FUNCTION_BLOCK "Graph_Sequence"   // FB265, GRAPH
VERSION : 0.1
// stored: AcknowledgeErrorsRequired true, AutoNumber true, GraphVersion 6.0, InitialValuesAcquisition false, IsIECCheckEnabled false, LanguageInNetworks LAD, LockOperatingMode false, PermanentILProcessingInMANMode false, SetENOAutomatically false, SkipSteps true, UDAEnableTagReadback false, WithAlarmHandling true
   // inherited from GRAPH_BASE
   VAR
      OFF_SQ_BASE : Bool;
   END_VAR
   VAR_INPUT
      ACK_EF { ExternalAccessible := 'False'; ExternalVisible := 'False'; ExternalWritable := 'False'} : Bool := false;   // Acknowledge all errors and faults
      INIT_SQ { ExternalAccessible := 'False'; ExternalVisible := 'False'; ExternalWritable := 'False'} : Bool := false;   // Set sequence to initial state
      stepTimeOutTime : Time;
      iInstance_Index : DInt;
   END_VAR
   VAR_IN_OUT
      funcGrp : "typeCaCgFg";   // Funktionsgruppe / Function Group
      fgControlGeneral_1 : "typeFgControlGeneral";   // Funktionsgruppe Steuerung / Function group control system
      ioJobSelect : Int;
   END_VAR
   VAR
      instGraphEval { ExternalAccessible := 'False'; ExternalVisible := 'False'; ExternalWritable := 'False'} : "GraphEvaluation";   // FG Laser 1: S7-Graph Auswertung / FG laser 1: S7-Graph evaluation
      fgControlGeneral { ExternalAccessible := 'False'; ExternalVisible := 'False'; ExternalWritable := 'False'} : "typeFgControlGeneral";   // Funktionsgruppe Steuerung / Function group control system
      stepTimeOut : Bool;
   END_VAR
BEGIN
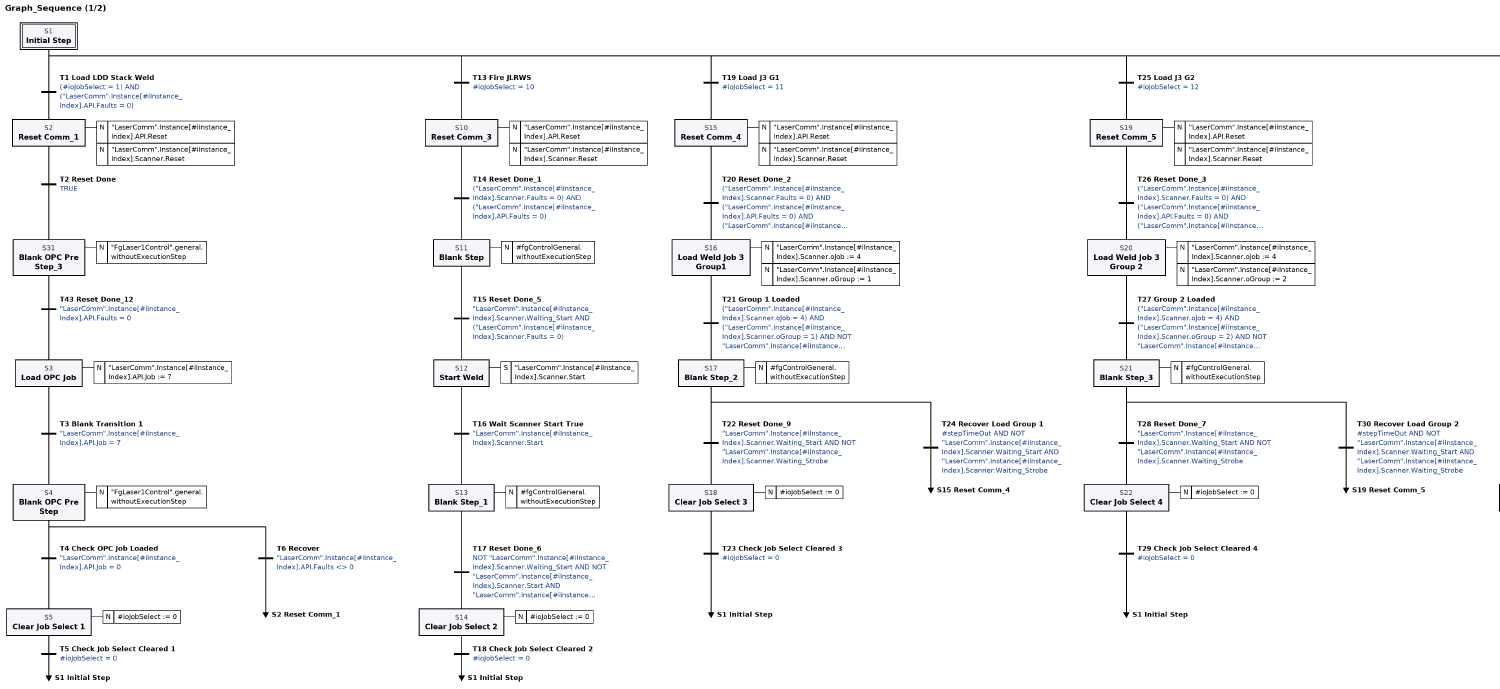
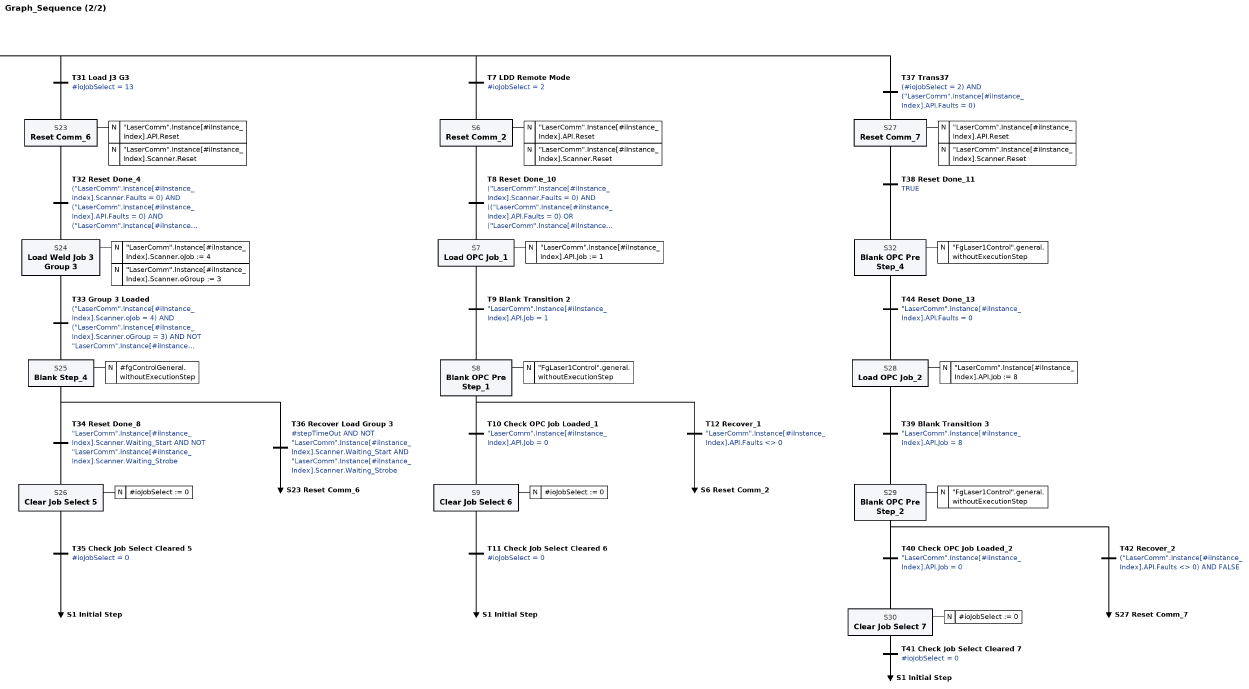
   // sequencer 1: Weld Graph Sequences
   INITIAL_STEP "Initial Step":   // S1, max time T#10S, warning time T#7S
   END_STEP
   TRANSITION "Load LDD Stack Weld" FROM "Initial Step" TO "Reset Comm_1"   // T1
      := (#ioJobSelect = 1) AND ("LaserComm".Instance[#iInstance_Index].API.Faults = 0);
   END_TRANSITION
   TRANSITION "Fire JLRWS" FROM "Initial Step" TO "Reset Comm_3"   // T13
      := #ioJobSelect = 10;
   END_TRANSITION
   TRANSITION "Load J3 G1" FROM "Initial Step" TO "Reset Comm_4"   // T19
      := #ioJobSelect = 11;
   END_TRANSITION
   TRANSITION "Load J3 G2" FROM "Initial Step" TO "Reset Comm_5"   // T25
      := #ioJobSelect = 12;
   END_TRANSITION
   TRANSITION "Load J3 G3" FROM "Initial Step" TO "Reset Comm_6"   // T31
      := #ioJobSelect = 13;
   END_TRANSITION
   TRANSITION "LDD Remote Mode" FROM "Initial Step" TO "Reset Comm_2"   // T7
      := #ioJobSelect = 2;
   END_TRANSITION
   TRANSITION Trans37 FROM "Initial Step" TO "Reset Comm_7"   // T37
      := (#ioJobSelect = 2) AND ("LaserComm".Instance[#iInstance_Index].API.Faults = 0);
   END_TRANSITION
   STEP "Reset Comm_1":   // S2, max time T#10S, warning time T#7S
      supervision V := #stepTimeOut;
              N    "LaserComm".Instance[#iInstance_Index].API.Reset
              N    "LaserComm".Instance[#iInstance_Index].Scanner.Reset
   END_STEP
   TRANSITION "Reset Done" FROM "Reset Comm_1" TO "Blank OPC Pre Step_3"   // T2
      := TRUE;
   END_TRANSITION
   STEP "Blank Step":   // S11, max time T#10S, warning time T#7S
      supervision V := #stepTimeOut;
              N    #fgControlGeneral.withoutExecutionStep
   END_STEP
   TRANSITION "Reset Done_5" FROM "Blank Step" TO "Start Weld"   // T15
      := "LaserComm".Instance[#iInstance_Index].Scanner.Waiting_Start AND ("LaserComm".Instance[#iInstance_Index].Scanner.Faults = 0);
   END_TRANSITION
   STEP "Clear Job Select 4":   // S22, max time T#10S, warning time T#7S
      supervision V := #stepTimeOut;
      // Clear Job Select
              N    #ioJobSelect := 0
   END_STEP
   TRANSITION "Check Job Select Cleared 4" FROM "Clear Job Select 4" TO "Initial Step"   // T29, jump: Check Jo Select Cleared
      := #ioJobSelect = 0;
   END_TRANSITION
   STEP "Clear Job Select 5":   // S26, max time T#10S, warning time T#7S
      supervision V := #stepTimeOut;
      // Clear Job Select
              N    #ioJobSelect := 0
   END_STEP
   TRANSITION "Check Job Select Cleared 5" FROM "Clear Job Select 5" TO "Initial Step"   // T35, jump: Check Jo Select Cleared
      := #ioJobSelect = 0;
   END_TRANSITION
   STEP "Load Weld Job 3 Group 3":   // S24, max time T#10S, warning time T#7S
      supervision V := #stepTimeOut;
              N    "LaserComm".Instance[#iInstance_Index].Scanner.oJob := 4
              N    "LaserComm".Instance[#iInstance_Index].Scanner.oGroup := 3
   END_STEP
   TRANSITION "Group 3 Loaded" FROM "Load Weld Job 3 Group 3" TO "Blank Step_4"   // T33
      := ("LaserComm".Instance[#iInstance_Index].Scanner.oJob = 4) AND ("LaserComm".Instance[#iInstance_Index].Scanner.oGroup = 3) AND NOT "LaserComm".Instance[#iInstance_Index].Scanner.Waiting_Strobe;
   END_TRANSITION
   STEP "Load OPC Job":   // S3, max time T#10S, warning time T#7S
      supervision V := #stepTimeOut;
              N    "LaserComm".Instance[#iInstance_Index].API.Job := 7
   END_STEP
   TRANSITION "Blank Transition 1" FROM "Load OPC Job" TO "Blank OPC Pre Step"   // T3
      := "LaserComm".Instance[#iInstance_Index].API.Job = 7;
   END_TRANSITION
   STEP "Blank OPC Pre Step":   // S4, max time T#10S, warning time T#7S
      supervision V := #stepTimeOut;
              N    "FgLaser1Control".general.withoutExecutionStep
   END_STEP
   TRANSITION "Check OPC Job Loaded" FROM "Blank OPC Pre Step" TO "Clear Job Select 1"   // T4
      := "LaserComm".Instance[#iInstance_Index].API.Job = 0;
   END_TRANSITION
   TRANSITION Recover FROM "Blank OPC Pre Step" TO "Reset Comm_1"   // T6, jump
      := "LaserComm".Instance[#iInstance_Index].API.Faults <> 0;
   END_TRANSITION
   STEP "Clear Job Select 1":   // S5, max time T#10S, warning time T#7S
      supervision V := #stepTimeOut;
      // Clear Job Select
              N    #ioJobSelect := 0
   END_STEP
   TRANSITION "Check Job Select Cleared 1" FROM "Clear Job Select 1" TO "Initial Step"   // T5, jump: Check Jo Select Cleared
      := #ioJobSelect = 0;
   END_TRANSITION
   STEP "Blank Step_1":   // S13, max time T#10S, warning time T#7S
      supervision V := #stepTimeOut;
              N    #fgControlGeneral.withoutExecutionStep
   END_STEP
   TRANSITION "Reset Done_6" FROM "Blank Step_1" TO "Clear Job Select 2"   // T17
      := NOT "LaserComm".Instance[#iInstance_Index].Scanner.Waiting_Start AND NOT "LaserComm".Instance[#iInstance_Index].Scanner.Start AND "LaserComm".Instance[#iInstance_Index].Scanner.Waiting_Strobe AND ("LaserComm".Instance[#iInstance_Index].Scanner.Faults = 0);
   END_TRANSITION
   STEP "Reset Comm_3":   // S10, max time T#10S, warning time T#7S
      supervision V := #stepTimeOut;
              N    "LaserComm".Instance[#iInstance_Index].API.Reset
              N    "LaserComm".Instance[#iInstance_Index].Scanner.Reset
   END_STEP
   TRANSITION "Reset Done_1" FROM "Reset Comm_3" TO "Blank Step"   // T14
      := ("LaserComm".Instance[#iInstance_Index].Scanner.Faults = 0) AND ("LaserComm".Instance[#iInstance_Index].API.Faults = 0);
   END_TRANSITION
   STEP "Load Weld Job 3 Group1":   // S16, max time T#10S, warning time T#7S
      supervision V := #stepTimeOut;
              N    "LaserComm".Instance[#iInstance_Index].Scanner.oJob := 4
              N    "LaserComm".Instance[#iInstance_Index].Scanner.oGroup := 1
   END_STEP
   TRANSITION "Group 1 Loaded" FROM "Load Weld Job 3 Group1" TO "Blank Step_2"   // T21
      := ("LaserComm".Instance[#iInstance_Index].Scanner.oJob = 4) AND ("LaserComm".Instance[#iInstance_Index].Scanner.oGroup = 1) AND NOT "LaserComm".Instance[#iInstance_Index].Scanner.Waiting_Strobe;
   END_TRANSITION
   STEP "Load Weld Job 3 Group 2":   // S20, max time T#10S, warning time T#7S
      supervision V := #stepTimeOut;
              N    "LaserComm".Instance[#iInstance_Index].Scanner.oJob := 4
              N    "LaserComm".Instance[#iInstance_Index].Scanner.oGroup := 2
   END_STEP
   TRANSITION "Group 2 Loaded" FROM "Load Weld Job 3 Group 2" TO "Blank Step_3"   // T27
      := ("LaserComm".Instance[#iInstance_Index].Scanner.oJob = 4) AND ("LaserComm".Instance[#iInstance_Index].Scanner.oGroup = 2) AND NOT "LaserComm".Instance[#iInstance_Index].Scanner.Waiting_Strobe;
   END_TRANSITION
   STEP "Reset Comm_4":   // S15, max time T#10S, warning time T#7S
      supervision V := #stepTimeOut;
              N    "LaserComm".Instance[#iInstance_Index].API.Reset
              N    "LaserComm".Instance[#iInstance_Index].Scanner.Reset
   END_STEP
   TRANSITION "Reset Done_2" FROM "Reset Comm_4" TO "Load Weld Job 3 Group1"   // T20
      := ("LaserComm".Instance[#iInstance_Index].Scanner.Faults = 0) AND ("LaserComm".Instance[#iInstance_Index].API.Faults = 0) AND ("LaserComm".Instance[#iInstance_Index].Scanner.oJob = 0) AND ("LaserComm".Instance[#iInstance_Index].Scanner.oGroup = 0) AND "LaserComm".Instance[#iInstance_Index].Scanner.Waiting_Strobe;
   END_TRANSITION
   STEP "Reset Comm_5":   // S19, max time T#10S, warning time T#7S
      supervision V := #stepTimeOut;
              N    "LaserComm".Instance[#iInstance_Index].API.Reset
              N    "LaserComm".Instance[#iInstance_Index].Scanner.Reset
   END_STEP
   TRANSITION "Reset Done_3" FROM "Reset Comm_5" TO "Load Weld Job 3 Group 2"   // T26
      := ("LaserComm".Instance[#iInstance_Index].Scanner.Faults = 0) AND ("LaserComm".Instance[#iInstance_Index].API.Faults = 0) AND ("LaserComm".Instance[#iInstance_Index].Scanner.oJob = 0) AND ("LaserComm".Instance[#iInstance_Index].Scanner.oGroup = 0);
   END_TRANSITION
   STEP "Reset Comm_6":   // S23, max time T#10S, warning time T#7S
      supervision V := #stepTimeOut;
              N    "LaserComm".Instance[#iInstance_Index].API.Reset
              N    "LaserComm".Instance[#iInstance_Index].Scanner.Reset
   END_STEP
   TRANSITION "Reset Done_4" FROM "Reset Comm_6" TO "Load Weld Job 3 Group 3"   // T32
      := ("LaserComm".Instance[#iInstance_Index].Scanner.Faults = 0) AND ("LaserComm".Instance[#iInstance_Index].API.Faults = 0) AND ("LaserComm".Instance[#iInstance_Index].Scanner.oJob = 0) AND ("LaserComm".Instance[#iInstance_Index].Scanner.oGroup = 0);
   END_TRANSITION
   STEP "Clear Job Select 3":   // S18, max time T#10S, warning time T#7S
      supervision V := #stepTimeOut;
      // Clear Job Select
              N    #ioJobSelect := 0
   END_STEP
   TRANSITION "Check Job Select Cleared 3" FROM "Clear Job Select 3" TO "Initial Step"   // T23, jump: Check Jo Select Cleared
      := #ioJobSelect = 0;
   END_TRANSITION
   STEP "Clear Job Select 2":   // S14, max time T#10S, warning time T#7S
      supervision V := #stepTimeOut;
      // Clear Job Select
              N    #ioJobSelect := 0
   END_STEP
   TRANSITION "Check Job Select Cleared 2" FROM "Clear Job Select 2" TO "Initial Step"   // T18, jump: Check Jo Select Cleared
      := #ioJobSelect = 0;
   END_TRANSITION
   STEP "Start Weld":   // S12, max time T#10S, warning time T#7S
      supervision V := #stepTimeOut;
              S    "LaserComm".Instance[#iInstance_Index].Scanner.Start
   END_STEP
   TRANSITION "Wait Scanner Start True" FROM "Start Weld" TO "Blank Step_1"   // T16
      := "LaserComm".Instance[#iInstance_Index].Scanner.Start;
   END_TRANSITION
   STEP "Blank Step_3":   // S21, max time T#10S, warning time T#7S
      supervision V := #stepTimeOut;
              N    #fgControlGeneral.withoutExecutionStep
   END_STEP
   TRANSITION "Reset Done_7" FROM "Blank Step_3" TO "Clear Job Select 4"   // T28
      := "LaserComm".Instance[#iInstance_Index].Scanner.Waiting_Start AND NOT "LaserComm".Instance[#iInstance_Index].Scanner.Waiting_Strobe;
   END_TRANSITION
   TRANSITION "Recover Load Group 2" FROM "Blank Step_3" TO "Reset Comm_5"   // T30, jump
      := #stepTimeOut AND NOT "LaserComm".Instance[#iInstance_Index].Scanner.Waiting_Start AND "LaserComm".Instance[#iInstance_Index].Scanner.Waiting_Strobe;
   END_TRANSITION
   STEP "Blank Step_4":   // S25, max time T#10S, warning time T#7S
      supervision V := #stepTimeOut;
              N    #fgControlGeneral.withoutExecutionStep
   END_STEP
   TRANSITION "Reset Done_8" FROM "Blank Step_4" TO "Clear Job Select 5"   // T34
      := "LaserComm".Instance[#iInstance_Index].Scanner.Waiting_Start AND NOT "LaserComm".Instance[#iInstance_Index].Scanner.Waiting_Strobe;
   END_TRANSITION
   TRANSITION "Recover Load Group 3" FROM "Blank Step_4" TO "Reset Comm_6"   // T36, jump
      := #stepTimeOut AND NOT "LaserComm".Instance[#iInstance_Index].Scanner.Waiting_Start AND "LaserComm".Instance[#iInstance_Index].Scanner.Waiting_Strobe;
   END_TRANSITION
   STEP "Blank Step_2":   // S17, max time T#10S, warning time T#7S
      supervision V := #stepTimeOut;
              N    #fgControlGeneral.withoutExecutionStep
   END_STEP
   TRANSITION "Reset Done_9" FROM "Blank Step_2" TO "Clear Job Select 3"   // T22
      := "LaserComm".Instance[#iInstance_Index].Scanner.Waiting_Start AND NOT "LaserComm".Instance[#iInstance_Index].Scanner.Waiting_Strobe;
   END_TRANSITION
   TRANSITION "Recover Load Group 1" FROM "Blank Step_2" TO "Reset Comm_4"   // T24, jump
      := #stepTimeOut AND NOT "LaserComm".Instance[#iInstance_Index].Scanner.Waiting_Start AND "LaserComm".Instance[#iInstance_Index].Scanner.Waiting_Strobe;
   END_TRANSITION
   STEP "Reset Comm_2":   // S6, max time T#10S, warning time T#7S
      supervision V := #stepTimeOut;
              N    "LaserComm".Instance[#iInstance_Index].API.Reset
              N    "LaserComm".Instance[#iInstance_Index].Scanner.Reset
   END_STEP
   TRANSITION "Reset Done_10" FROM "Reset Comm_2" TO "Load OPC Job_1"   // T8
      := ("LaserComm".Instance[#iInstance_Index].Scanner.Faults = 0) AND (("LaserComm".Instance[#iInstance_Index].API.Faults = 0) OR ("LaserComm".Instance[#iInstance_Index].API.Faults = 64));
   END_TRANSITION
   STEP "Load OPC Job_1":   // S7, max time T#10S, warning time T#7S
      supervision V := #stepTimeOut;
              N    "LaserComm".Instance[#iInstance_Index].API.Job := 1
   END_STEP
   TRANSITION "Blank Transition 2" FROM "Load OPC Job_1" TO "Blank OPC Pre Step_1"   // T9
      := "LaserComm".Instance[#iInstance_Index].API.Job = 1;
   END_TRANSITION
   STEP "Blank OPC Pre Step_1":   // S8, max time T#10S, warning time T#7S
      supervision V := #stepTimeOut;
              N    "FgLaser1Control".general.withoutExecutionStep
   END_STEP
   TRANSITION "Check OPC Job Loaded_1" FROM "Blank OPC Pre Step_1" TO "Clear Job Select 6"   // T10
      := "LaserComm".Instance[#iInstance_Index].API.Job = 0;
   END_TRANSITION
   TRANSITION Recover_1 FROM "Blank OPC Pre Step_1" TO "Reset Comm_2"   // T12, jump
      := "LaserComm".Instance[#iInstance_Index].API.Faults <> 0;
   END_TRANSITION
   STEP "Clear Job Select 6":   // S9, max time T#10S, warning time T#7S
      supervision V := #stepTimeOut;
      // Clear Job Select
              N    #ioJobSelect := 0
   END_STEP
   TRANSITION "Check Job Select Cleared 6" FROM "Clear Job Select 6" TO "Initial Step"   // T11, jump: Check Jo Select Cleared
      := #ioJobSelect = 0;
   END_TRANSITION
   STEP "Reset Comm_7":   // S27, max time T#10S, warning time T#7S
      supervision V := #stepTimeOut;
              N    "LaserComm".Instance[#iInstance_Index].API.Reset
              N    "LaserComm".Instance[#iInstance_Index].Scanner.Reset
   END_STEP
   TRANSITION "Reset Done_11" FROM "Reset Comm_7" TO "Blank OPC Pre Step_4"   // T38
      := TRUE;
   END_TRANSITION
   STEP "Load OPC Job_2":   // S28, max time T#10S, warning time T#7S
      supervision V := #stepTimeOut;
              N    "LaserComm".Instance[#iInstance_Index].API.Job := 8
   END_STEP
   TRANSITION "Blank Transition 3" FROM "Load OPC Job_2" TO "Blank OPC Pre Step_2"   // T39
      := "LaserComm".Instance[#iInstance_Index].API.Job = 8;
   END_TRANSITION
   STEP "Blank OPC Pre Step_2":   // S29, max time T#10S, warning time T#7S
      supervision V := #stepTimeOut;
              N    "FgLaser1Control".general.withoutExecutionStep
   END_STEP
   TRANSITION "Check OPC Job Loaded_2" FROM "Blank OPC Pre Step_2" TO "Clear Job Select 7"   // T40
      := "LaserComm".Instance[#iInstance_Index].API.Job = 0;
   END_TRANSITION
   TRANSITION Recover_2 FROM "Blank OPC Pre Step_2" TO "Reset Comm_7"   // T42, jump
      := ("LaserComm".Instance[#iInstance_Index].API.Faults <> 0) AND FALSE;
   END_TRANSITION
   STEP "Clear Job Select 7":   // S30, max time T#10S, warning time T#7S
      supervision V := #stepTimeOut;
      // Clear Job Select
              N    #ioJobSelect := 0
   END_STEP
   TRANSITION "Check Job Select Cleared 7" FROM "Clear Job Select 7" TO "Initial Step"   // T41, jump: Check Jo Select Cleared
      := #ioJobSelect = 0;
   END_TRANSITION
   STEP "Blank OPC Pre Step_3":   // S31, max time T#10S, warning time T#7S
      supervision V := #stepTimeOut;
              N    "FgLaser1Control".general.withoutExecutionStep
   END_STEP
   TRANSITION "Reset Done_12" FROM "Blank OPC Pre Step_3" TO "Load OPC Job"   // T43
      := "LaserComm".Instance[#iInstance_Index].API.Faults = 0;
   END_TRANSITION
   STEP "Blank OPC Pre Step_4":   // S32, max time T#10S, warning time T#7S
      supervision V := #stepTimeOut;
              N    "FgLaser1Control".general.withoutExecutionStep
   END_STEP
   TRANSITION "Reset Done_13" FROM "Blank OPC Pre Step_4" TO "Load OPC Job_2"   // T44
      := "LaserComm".Instance[#iInstance_Index].API.Faults = 0;
   END_TRANSITION

   // permanent post-instructions
   NETWORK 1
      #instGraphEval(rtData := #RT_DATA,   // "GraphEvaluation"
                     timeOutTime := #stepTimeOutTime,
                     funcGrp := #funcGrp,
                     fgControlGeneral := #fgControlGeneral,
                     timeOut => #stepTimeOut);
END_FUNCTION_BLOCK

FUNCTION_BLOCK "GraphEvaluation"   // FB38, LAD
TITLE = S7 graph evaluation / S7-Graph Auswertung
{ S7_Optimized_Access := 'TRUE' }
AUTHOR : Grob
FAMILY : Kernel_V2
VERSION : 1.4
// S7 graph evaluation / S7-Graph Auswertung
// stored: AutoNumber true, IsIECCheckEnabled true, IsRetainMemResEnabled false, MemoryReserve 100, SetENOAutomatically true, UDAEnableTagReadback false
   VAR_INPUT
      rtData { ExternalAccessible := 'False'; ExternalVisible := 'False'; ExternalWritable := 'False'} : G7_RTDataPlus_V6;   // Graph RT_DATA
      timeOutTime { ExternalAccessible := 'False'; ExternalVisible := 'False'; ExternalWritable := 'False'} : Time := T#5m;   // Timeout Zeit / Timeout time
   END_VAR
   VAR_OUTPUT
      timeOut { ExternalAccessible := 'False'; ExternalVisible := 'False'; ExternalWritable := 'False'} : Bool;   // Timeout Fehler / Timeout error
   END_VAR
   VAR_IN_OUT
      funcGrp : "typeCaCgFg";   // Funktionsgruppe / Function Group
      fgControlGeneral : "typeFgControlGeneral";   // Funktionsgruppe Allgemeine Steuerschnittstelle / General control interface function group
   END_VAR
   VAR
      statErrorTimeOut { ExternalAccessible := 'False'; ExternalVisible := 'False'; ExternalWritable := 'False'} : Bool;   // ProDiag-Störung: Timeout / ProDiag fault: Timeout
      statCount { ExternalAccessible := 'False'; ExternalVisible := 'False'; ExternalWritable := 'False'} : USInt;   // Zähler / Counter
      statFgName { ExternalAccessible := 'False'; ExternalVisible := 'False'; ExternalWritable := 'False'} : WString["GRP_JOB_NAME_SIZE"];   // ProDiag Begleitwert: Name der FG / ProDiag associated value: Name of the FG
      statGraphStepNumber { ExternalAccessible := 'False'; ExternalVisible := 'False'; ExternalWritable := 'False'} : Int;   // ProDiag Begleitwert: Schrittnummer / ProDiag associated value: step number
      statLastStepNumber { ExternalAccessible := 'False'; ExternalVisible := 'False'; ExternalWritable := 'False'} : Int;   // Letzte Schrittnummer gespeichert / Last step number saved
      instTimerTimeOut { ExternalAccessible := 'False'; ExternalVisible := 'False'; ExternalWritable := 'False'} : TON_TIME;   // Timer Timeout / Timer for timeout
   END_VAR
BEGIN

REGION Network 1 (SCL): Version
   //===============================================================================================================================
   // GROB-WERKE GmbH & Co. KG
   // (c)Copyright 2022 All Rights Reserved
   //
   // Reproduction, replication, modification, distribution, communication to the public and making the work available to the public
   // or others as well as other exploitation of the software and, if applicable, the medium containing the software without express
   // authorization is prohibited. Offenders will be held liable for the payment of damages. All rights reserved with regard to the
   // protection of intellectual property
   // ------------------------------------------------------------------------------------------------------------------------------
   //     Library:       Kernel V2
   //     Tested with:   PLCSIM
   //     Engineering:   TIA Portal V17
   //     Restrictions:  ---
   //     Requirements:  ---
   REGION Functionality
       //                This function block has to be  called in the permanent post-instructions
       //
       //                It evaluates information of the graph and writes informations to the function group
       //                control interface (typeFgControlGeneral in Fg*General-DB)
       //                Further it triggers stop to the function group in single step mode after finishing a sequence step
       //
       //                Handles the general graph step time out
   END_REGION
   // ------------------------------------------------------------------------------------------------------------------------------
   // Change log table: 
   //     Version    Date      Expert in charge    Changes applied 
   //     -------|------------|-----------------|-----------------------------------------------------------------------------------
   //     00.00    24.05.2022  Dorn, F.            Migrated from TST V1.4, block version 01.00
   //     01.00    24.05.2022  Dorn, F.            First released version
   //     01.01    02.08.2022  Dorn, F.            Reset functiongroup after graph reinitialization
   //     01.02    21.11.2022  Dorn, F.            Fixed graph time out. (caused 2 alarms)
   //     01.03    18.02.2023  Dorn, F.            Implemented new internal signals in typeFgControlGeneral 
   //                                                  (start delays for GraphControl-funciton)
   //     01.04    18.12.2023  Dorn, F.            Implemented signals for stop selected by...
   //===============================================================================================================================
END_REGION

REGION Network 3: *************** General *************** / *************** Allgemein ***************
END_REGION

REGION Network 4: Graph fault sent to group / Graph Störung an Gruppe übertragen
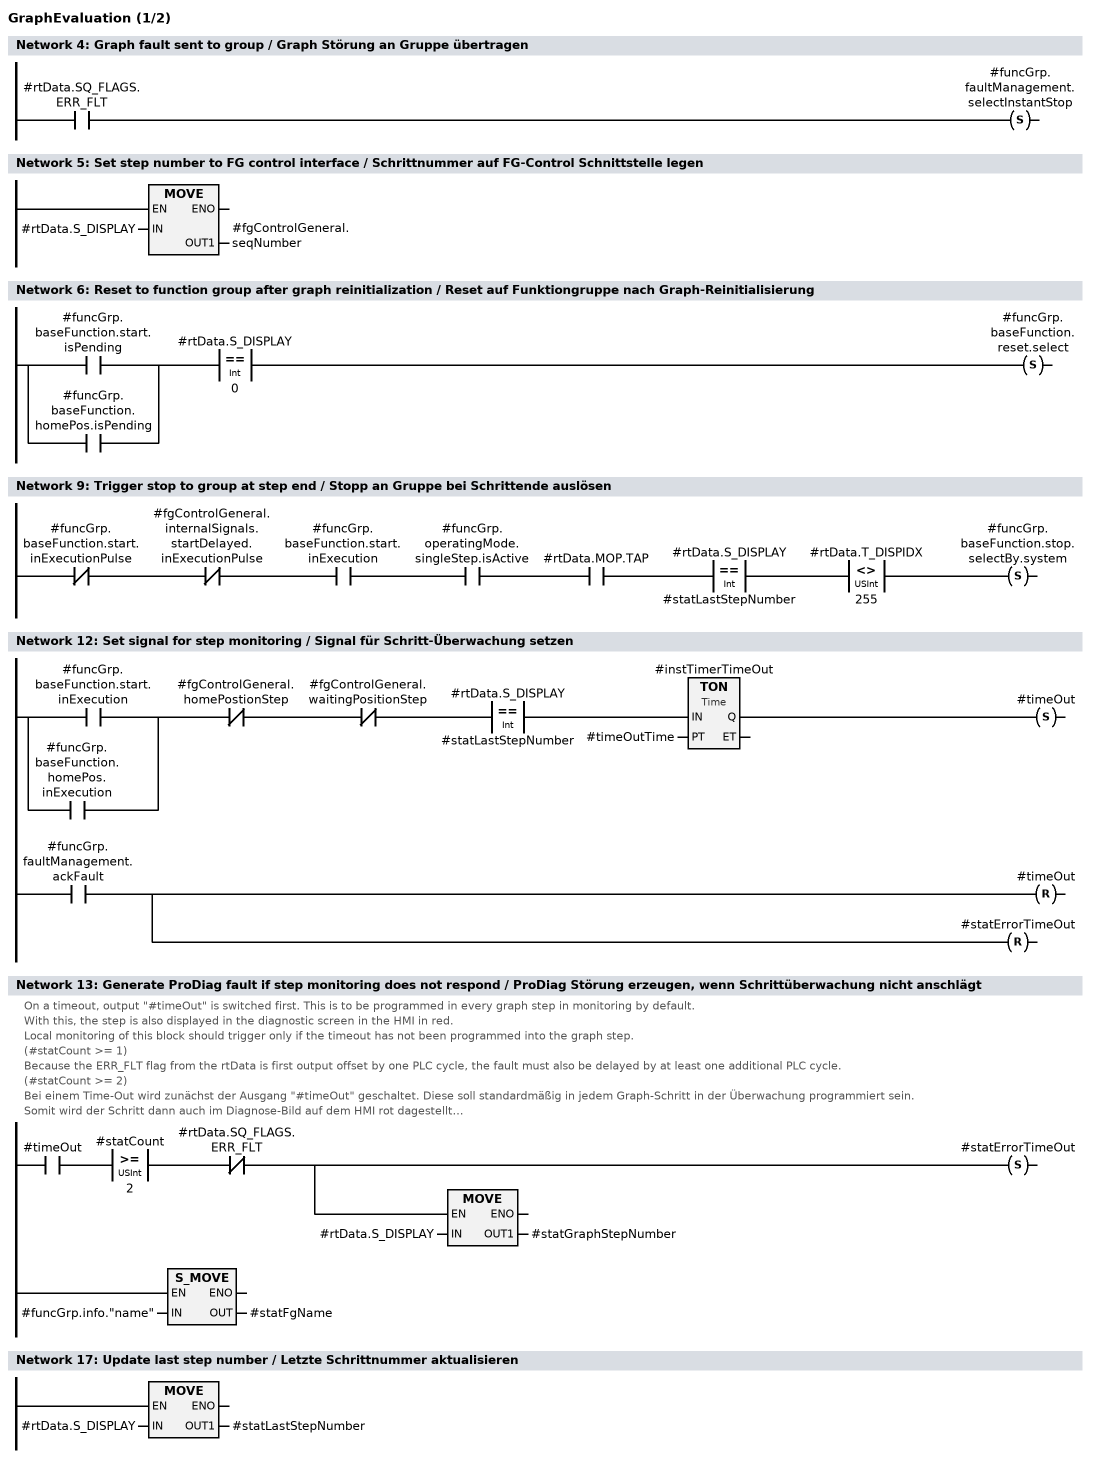
   RUNG wire#powerrail
      Contact( #rtData.SQ_FLAGS.ERR_FLT )
      S_Coil( #funcGrp.faultManagement.selectInstantStop )
   END_RUNG
   // the same network as SCL:
   IF #rtData.SQ_FLAGS.ERR_FLT THEN #funcGrp.faultManagement.selectInstantStop := TRUE; END_IF;
END_REGION

REGION Network 5: Set step number to FG control interface / Schrittnummer auf FG-Control Schnittstelle legen
   RUNG wire#powerrail
      Move(in := #rtData.S_DISPLAY, out1 => #fgControlGeneral.seqNumber)
   END_RUNG
   // the same network as SCL:
   #fgControlGeneral.seqNumber := #rtData.S_DISPLAY;
END_REGION

REGION Network 6: Reset to function group after graph reinitialization / Reset auf Funktiongruppe nach Graph-Reinitialisierung
   RUNG wire#powerrail
      Contact( #funcGrp.baseFunction.start.isPending )
      wire#w1
      { S7_Templates := "SrcType := Int" } EQ_Contact(in1 := #rtData.S_DISPLAY, in2 := 0)
      S_Coil( #funcGrp.baseFunction.reset.select )
   END_RUNG
   RUNG wire#powerrail
      Contact( #funcGrp.baseFunction.homePos.isPending )
   END_RUNG wire#w1
   // the same network as SCL:
   IF (#funcGrp.baseFunction.start.isPending OR #funcGrp.baseFunction.homePos.isPending) AND (#rtData.S_DISPLAY = 0) THEN
       #funcGrp.baseFunction.reset.select := TRUE;
   END_IF;
END_REGION

REGION Network 8: *************** Single-step (TAP) *************** / *************** Einzelschritt (TAP) ***************
END_REGION

REGION Network 9: Trigger stop to group at step end / Stopp an Gruppe bei Schrittende auslösen
   RUNG wire#powerrail
      I_Contact( #funcGrp.baseFunction.start.inExecutionPulse )
      I_Contact( #fgControlGeneral.internalSignals.startDelayed.inExecutionPulse )
      Contact( #funcGrp.baseFunction.start.inExecution )
      Contact( #funcGrp.operatingMode.singleStep.isActive )
      Contact( #rtData.MOP.TAP )
      { S7_Templates := "SrcType := Int" } EQ_Contact(in1 := #rtData.S_DISPLAY, in2 := #statLastStepNumber)
      { S7_Templates := "SrcType := USInt" } NE_Contact(in1 := #rtData.T_DISPIDX, in2 := 255)
      S_Coil( #funcGrp.baseFunction.stop.selectBy.system )
   END_RUNG
   // the same network as SCL:
   IF NOT #funcGrp.baseFunction.start.inExecutionPulse AND NOT #fgControlGeneral.internalSignals.startDelayed.inExecutionPulse AND #funcGrp.baseFunction.start.inExecution AND #funcGrp.operatingMode.singleStep.isActive AND #rtData.MOP.TAP AND (#rtData.S_DISPLAY = #statLastStepNumber) AND (#rtData.T_DISPIDX <> 255) THEN
       #funcGrp.baseFunction.stop.selectBy.system := TRUE;
   END_IF;
END_REGION

REGION Network 11: *************** Timeout monitoring *************** / *************** Timeout Überwachung ***************
END_REGION

REGION Network 12: Set signal for step monitoring / Signal für Schritt-Überwachung setzen
   RUNG wire#powerrail
      Contact( #funcGrp.baseFunction.start.inExecution )
      wire#w1
      I_Contact( #fgControlGeneral.homePostionStep )
      I_Contact( #fgControlGeneral.waitingPositionStep )
      { S7_Templates := "SrcType := Int" } EQ_Contact(in1 := #rtData.S_DISPLAY, in2 := #statLastStepNumber)
      { S7_Templates := "time_type := Time" } #instTimerTimeOut.TON(pt := #timeOutTime, et =>)
      S_Coil( #timeOut )
   END_RUNG
   RUNG wire#powerrail
      Contact( #funcGrp.baseFunction.homePos.inExecution )
   END_RUNG wire#w1
   RUNG wire#powerrail
      Contact( #funcGrp.faultManagement.ackFault )
      wire#w2
      R_Coil( #timeOut )
   END_RUNG
   RUNG wire#w2
      R_Coil( #statErrorTimeOut )
   END_RUNG
   // the same network as SCL:
   #instTimerTimeOut(IN := (#funcGrp.baseFunction.start.inExecution OR #funcGrp.baseFunction.homePos.inExecution) AND NOT #fgControlGeneral.homePostionStep AND NOT #fgControlGeneral.waitingPositionStep AND (#rtData.S_DISPLAY = #statLastStepNumber),   // TON
                     PT := #timeOutTime);
   IF #instTimerTimeOut.Q THEN #timeOut := TRUE; END_IF;
   IF #funcGrp.faultManagement.ackFault THEN
       #timeOut := FALSE;
       #statErrorTimeOut := FALSE;
   END_IF;
END_REGION

REGION Network 13: Generate ProDiag fault if step monitoring does not respond / ProDiag Störung erzeugen, wenn Schrittüberwachung nicht anschlägt
   // On a timeout, output "#timeOut" is switched first. This is to be programmed in every graph step in monitoring by default.
   // With this, the step is also displayed in the diagnostic screen in the HMI in red.
   // Local monitoring of this block should trigger only if the timeout has not been programmed into the graph step.
   // (#statCount >= 1)
   // 
   // Because the ERR_FLT flag from the rtData is first output offset by one PLC cycle, the fault must also be delayed by at least one additional PLC cycle.
   // (#statCount >= 2)
   // Bei einem Time-Out wird zunächst der Ausgang "#timeOut" geschaltet. Diese soll standardmäßig in jedem Graph-Schritt in der Überwachung programmiert sein.
   // Somit wird der Schritt dann auch im Diagnose-Bild auf dem HMI rot dagestellt.
   // Nur, wenn der Time-Out im Graphschritt nicht programmeirt wurde, soll die lokale Überwachung von diesem Baustein auslösen.
   // (#statCount >= 1)
   // 
   // Da das Flag ERR_FLT vom den rtData erst um einen PLC-Zyklus versetzt ausgegeben wird, muss die Störung zusätzlich noch um mindestens einen PLC-Zyklus  verzögert werden.
   // (#statCount >= 2)
   RUNG wire#powerrail
      Contact( #timeOut )
      { S7_Templates := "SrcType := USInt" } GE_Contact(in1 := #statCount, in2 := 2)
      I_Contact( #rtData.SQ_FLAGS.ERR_FLT )
      wire#w1
      S_Coil( #statErrorTimeOut )
   END_RUNG
   RUNG wire#w1
      Move(in := #rtData.S_DISPLAY, out1 => #statGraphStepNumber)
   END_RUNG
   RUNG wire#powerrail
      S_Move(in := #funcGrp.info."name", out => #statFgName)
   END_RUNG
   // the same network as SCL:
   IF #timeOut AND (#statCount >= 2) AND NOT #rtData.SQ_FLAGS.ERR_FLT THEN
       #statErrorTimeOut := TRUE;
       #statGraphStepNumber := #rtData.S_DISPLAY;
   END_IF;
   #statFgName := #funcGrp.info."name";
END_REGION

REGION Network 14 (SCL): Counter for fault / Zähler für Störung
   IF #timeOut AND NOT (#rtData.SQ_FLAGS.ERR_FLT OR #statErrorTimeOut) THEN
       #statCount += 1;
   ELSIF NOT #timeOut THEN
       #statCount := 0;
   END_IF;
END_REGION

REGION Network 16: *************** Internal control signals *************** / *************** Interne Steuersignale ***************
END_REGION

REGION Network 17: Update last step number / Letzte Schrittnummer aktualisieren
   RUNG wire#powerrail
      Move(in := #rtData.S_DISPLAY, out1 => #statLastStepNumber)
   END_RUNG
   // the same network as SCL:
   #statLastStepNumber := #rtData.S_DISPLAY;
END_REGION

REGION Network 18: Delayed start signals for "GraphControl"-FC / Verzögerte Start-Signale für "GraphControl"-FC
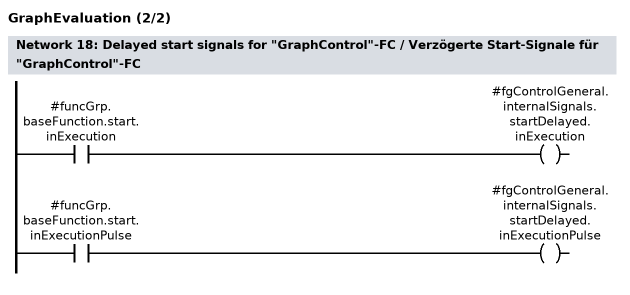
   RUNG wire#powerrail
      Contact( #funcGrp.baseFunction.start.inExecution )
      Coil( #fgControlGeneral.internalSignals.startDelayed.inExecution )
   END_RUNG
   RUNG wire#powerrail
      Contact( #funcGrp.baseFunction.start.inExecutionPulse )
      Coil( #fgControlGeneral.internalSignals.startDelayed.inExecutionPulse )
   END_RUNG
   // the same network as SCL:
   #fgControlGeneral.internalSignals.startDelayed.inExecution := #funcGrp.baseFunction.start.inExecution;
   #fgControlGeneral.internalSignals.startDelayed.inExecutionPulse := #funcGrp.baseFunction.start.inExecutionPulse;
END_REGION
END_FUNCTION_BLOCK

FUNCTION_BLOCK "Control"   // FB266, LAD
{ S7_Optimized_Access := 'FALSE' }
VERSION : 0.1
// stored: AutoNumber true, IsIECCheckEnabled false, SetENOAutomatically false, UDAEnableTagReadback false
   VAR_INPUT
      iGraph_Step_1 : Bool;
      iInstance_Index : DInt;
   END_VAR
   VAR_IN_OUT
      ioGraph_Job_Select : Int;
   END_VAR
   VAR DB_SPECIFIC
      sStep : DInt;
      sNo_Faults_Active : Bool;
      Step_Delay { S7_SetPoint := 'True'} : TON_TIME;
      sCounter_Done : Bool;
      sCTU : IEC_COUNTER;
      sWeldJob { S7_SetPoint := 'True'} : Byte;
      sDelayDone : Bool;
   END_VAR
   VAR_TEMP   // added for the SCL form of the ladder/FBD networks
      _w1 : Bool;
      _w2 : Bool;
   END_VAR
BEGIN

REGION Network 1: Tooling Delay
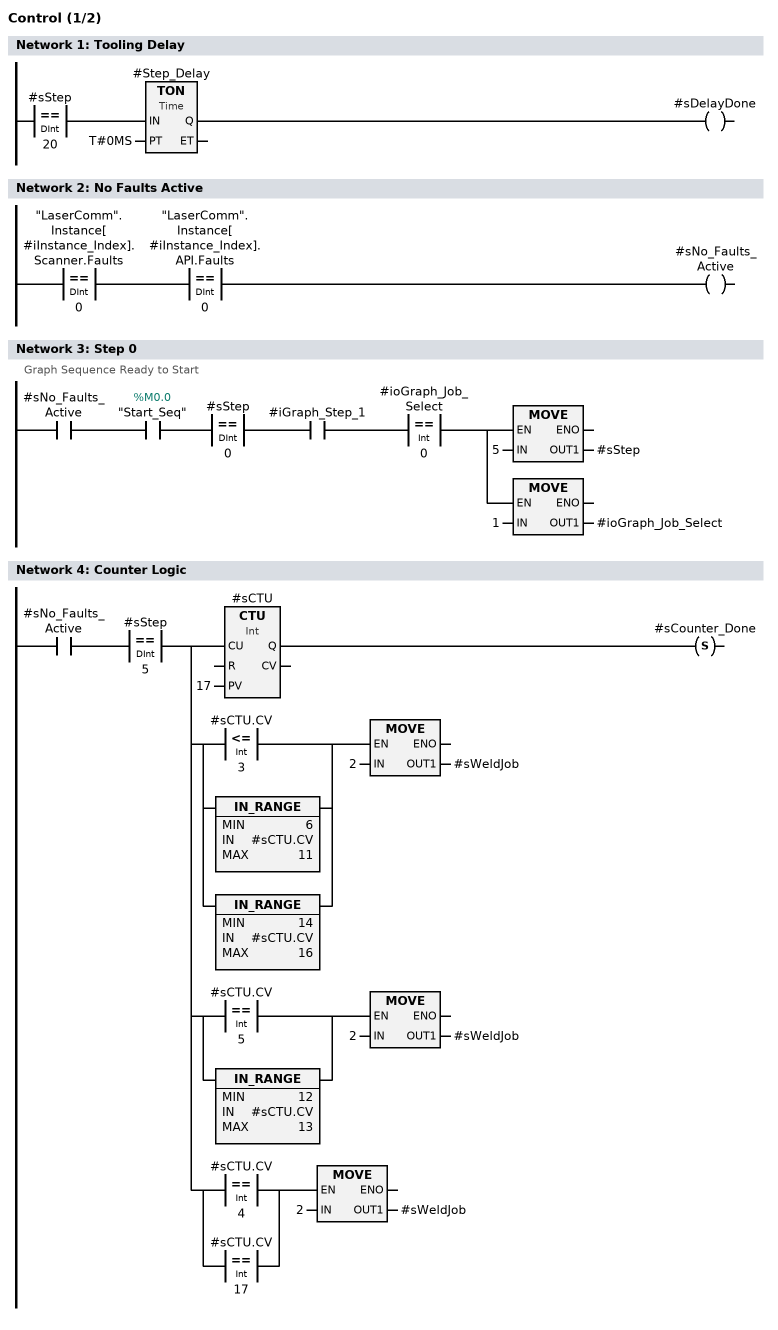
   RUNG wire#powerrail
      { S7_Templates := "SrcType := DInt" } EQ_Contact(in1 := #sStep, in2 := 20)
      { S7_Templates := "time_type := Time" } #Step_Delay.TON(pt := T#0MS, et =>)
      Coil( #sDelayDone )
   END_RUNG
   // the same network as SCL:
   #Step_Delay(IN := #sStep = 20, PT := T#0MS);   // TON
   #sDelayDone := #Step_Delay.Q;
END_REGION

REGION Network 2: No Faults Active
   RUNG wire#powerrail
      { S7_Templates := "SrcType := DInt" } EQ_Contact(in1 := "LaserComm".Instance[#iInstance_Index].Scanner.Faults, in2 := 0)
      { S7_Templates := "SrcType := DInt" } EQ_Contact(in1 := "LaserComm".Instance[#iInstance_Index].API.Faults, in2 := 0)
      Coil( #sNo_Faults_Active )
   END_RUNG
   // the same network as SCL:
   #sNo_Faults_Active := ("LaserComm".Instance[#iInstance_Index].Scanner.Faults = 0) AND ("LaserComm".Instance[#iInstance_Index].API.Faults = 0);
END_REGION

REGION Network 3: Step 0
   // Graph Sequence Ready to Start
   RUNG wire#powerrail
      Contact( #sNo_Faults_Active )
      Contact( "Start_Seq" )
      { S7_Templates := "SrcType := DInt" } EQ_Contact(in1 := #sStep, in2 := 0)
      Contact( #iGraph_Step_1 )
      { S7_Templates := "SrcType := Int" } EQ_Contact(in1 := #ioGraph_Job_Select, in2 := 0)
      wire#w1
      { S7_GenerateENO := "TRUE" } Move(in := 5, out1 => #sStep)
   END_RUNG
   RUNG wire#w1
      { S7_GenerateENO := "TRUE" } Move(in := 1, out1 => #ioGraph_Job_Select)
   END_RUNG
   // the same network as SCL:
   #_w1 := #sNo_Faults_Active AND "Start_Seq" AND (#sStep = 0) AND #iGraph_Step_1 AND (#ioGraph_Job_Select = 0);
   IF #_w1 THEN
       #sStep := 5;
       #ioGraph_Job_Select := 1;
   END_IF;
END_REGION

REGION Network 4: Counter Logic
   RUNG wire#powerrail
      Contact( #sNo_Faults_Active )
      { S7_Templates := "SrcType := DInt" } EQ_Contact(in1 := #sStep, in2 := 5)
      wire#w1
      { S7_Templates := "value_type := Int" } #sCTU.CTU(r :=, pv := 17, cv =>)
      S_Coil( #sCounter_Done )
   END_RUNG
   RUNG wire#w1
      { S7_Templates := "SrcType := Int" } LE_Contact(in1 := #sCTU.CV, in2 := 3)
      wire#w2
      Move(in := 2, out1 => #sWeldJob)
   END_RUNG
   RUNG wire#w1
      { S7_Templates := "SrcType := Int" } InRange(min := 6, in := #sCTU.CV, max := 11)
   END_RUNG wire#w2
   RUNG wire#w1
      { S7_Templates := "SrcType := Int" } InRange(min := 14, in := #sCTU.CV, max := 16)
   END_RUNG wire#w2
   RUNG wire#w1
      { S7_Templates := "SrcType := Int" } EQ_Contact(in1 := #sCTU.CV, in2 := 5)
      wire#w3
      Move(in := 2, out1 => #sWeldJob)
   END_RUNG
   RUNG wire#w1
      { S7_Templates := "SrcType := Int" } InRange(min := 12, in := #sCTU.CV, max := 13)
   END_RUNG wire#w3
   RUNG wire#w1
      { S7_Templates := "SrcType := Int" } EQ_Contact(in1 := #sCTU.CV, in2 := 4)
      wire#w4
      Move(in := 2, out1 => #sWeldJob)
   END_RUNG
   RUNG wire#w1
      { S7_Templates := "SrcType := Int" } EQ_Contact(in1 := #sCTU.CV, in2 := 17)
   END_RUNG wire#w4
   // the same network as SCL:
   #_w1 := #sNo_Faults_Active AND (#sStep = 5);
   #sCTU.CTU(CU := #_w1, PV := 17);
   IF #sCTU.Q THEN #sCounter_Done := TRUE; END_IF;
   IF #_w1 AND ((#sCTU.CV <= 3) OR ((6 <= #sCTU.CV) AND (#sCTU.CV <= 11)) OR ((14 <= #sCTU.CV) AND (#sCTU.CV <= 16))) THEN
       #sWeldJob := 2;
   END_IF;
   IF #_w1 AND ((#sCTU.CV = 5) OR ((12 <= #sCTU.CV) AND (#sCTU.CV <= 13))) THEN #sWeldJob := 2; END_IF;
   IF #_w1 AND ((#sCTU.CV = 4) OR (#sCTU.CV = 17)) THEN #sWeldJob := 2; END_IF;
END_REGION

REGION Network 5: Step 5
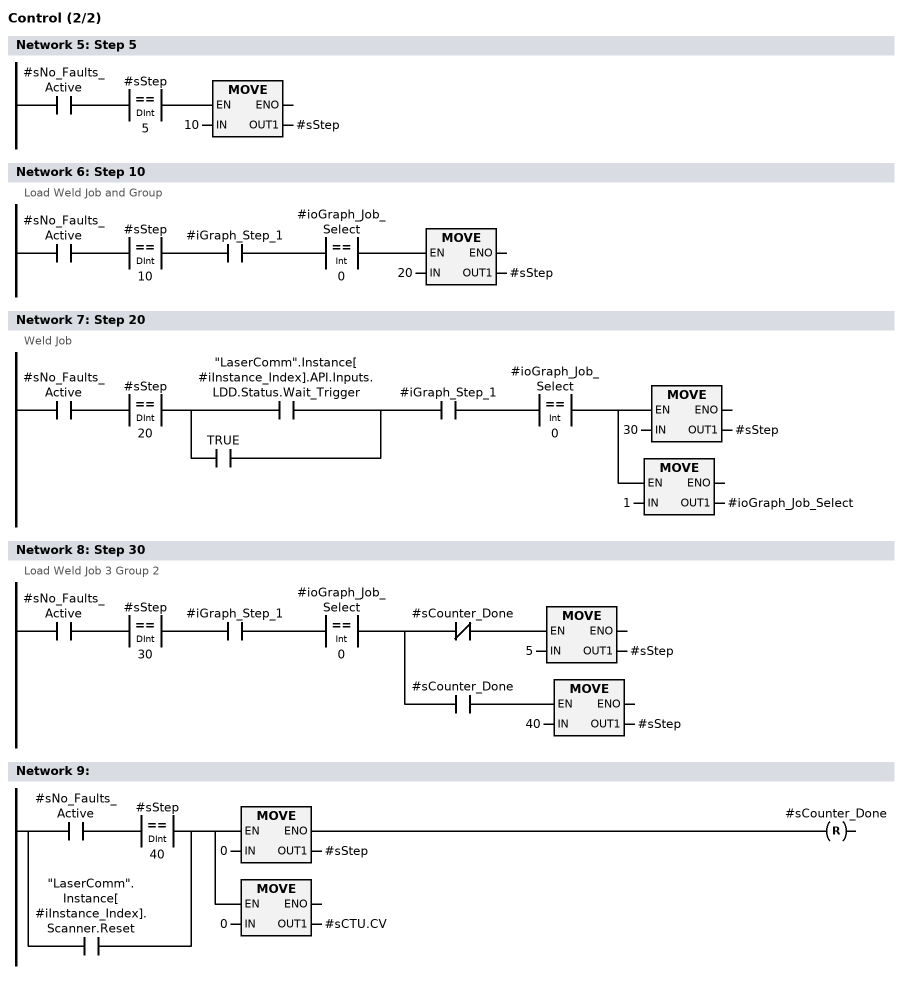
   RUNG wire#powerrail
      Contact( #sNo_Faults_Active )
      { S7_Templates := "SrcType := DInt" } EQ_Contact(in1 := #sStep, in2 := 5)
      { S7_GenerateENO := "TRUE" } Move(in := 10, out1 => #sStep)
   END_RUNG
   // the same network as SCL:
   IF #sNo_Faults_Active AND (#sStep = 5) THEN #sStep := 10; END_IF;
END_REGION

REGION Network 6: Step 10
   // Load Weld Job and Group
   RUNG wire#powerrail
      Contact( #sNo_Faults_Active )
      { S7_Templates := "SrcType := DInt" } EQ_Contact(in1 := #sStep, in2 := 10)
      Contact( #iGraph_Step_1 )
      { S7_Templates := "SrcType := Int" } EQ_Contact(in1 := #ioGraph_Job_Select, in2 := 0)
      { S7_GenerateENO := "TRUE" } Move(in := 20, out1 => #sStep)
   END_RUNG
   // the same network as SCL:
   IF #sNo_Faults_Active AND (#sStep = 10) AND #iGraph_Step_1 AND (#ioGraph_Job_Select = 0) THEN
       #sStep := 20;
   END_IF;
END_REGION

REGION Network 7: Step 20
   // Weld Job
   RUNG wire#powerrail
      Contact( #sNo_Faults_Active )
      { S7_Templates := "SrcType := DInt" } EQ_Contact(in1 := #sStep, in2 := 20)
      wire#w1
      Contact( "LaserComm".Instance[#iInstance_Index].API.Inputs.LDD.Status.Wait_Trigger )
      wire#w2
      Contact( #iGraph_Step_1 )
      { S7_Templates := "SrcType := Int" } EQ_Contact(in1 := #ioGraph_Job_Select, in2 := 0)
      wire#w3
      { S7_GenerateENO := "TRUE" } Move(in := 30, out1 => #sStep)
   END_RUNG
   RUNG wire#w1
      Contact( TRUE )
   END_RUNG wire#w2
   RUNG wire#w3
      { S7_GenerateENO := "TRUE" } Move(in := 1, out1 => #ioGraph_Job_Select)
   END_RUNG
   // the same network as SCL:
   #_w1 := #sNo_Faults_Active AND (#sStep = 20) AND ("LaserComm".Instance[#iInstance_Index].API.Inputs.LDD.Status.Wait_Trigger OR TRUE) AND #iGraph_Step_1 AND (#ioGraph_Job_Select = 0);
   IF #_w1 THEN
       #sStep := 30;
       #ioGraph_Job_Select := 1;
   END_IF;
END_REGION

REGION Network 8: Step 30
   // Load Weld Job 3 Group 2
   RUNG wire#powerrail
      Contact( #sNo_Faults_Active )
      { S7_Templates := "SrcType := DInt" } EQ_Contact(in1 := #sStep, in2 := 30)
      Contact( #iGraph_Step_1 )
      { S7_Templates := "SrcType := Int" } EQ_Contact(in1 := #ioGraph_Job_Select, in2 := 0)
      wire#w1
      I_Contact( #sCounter_Done )
      { S7_GenerateENO := "TRUE" } Move(in := 5, out1 => #sStep)
   END_RUNG
   RUNG wire#w1
      Contact( #sCounter_Done )
      { S7_GenerateENO := "TRUE" } Move(in := 40, out1 => #sStep)
   END_RUNG
   // the same network as SCL:
   #_w1 := #sNo_Faults_Active AND (#sStep = 30) AND #iGraph_Step_1 AND (#ioGraph_Job_Select = 0);
   IF #_w1 AND NOT #sCounter_Done THEN #sStep := 5; END_IF;
   IF #_w1 AND #sCounter_Done THEN #sStep := 40; END_IF;
END_REGION

REGION Network 9
   RUNG wire#powerrail
      Contact( #sNo_Faults_Active )
      { S7_Templates := "SrcType := DInt" } EQ_Contact(in1 := #sStep, in2 := 40)
      wire#w1
      { S7_GenerateENO := "TRUE" } Move(in := 0, out1 => #sStep)
      R_Coil( #sCounter_Done )
   END_RUNG
   RUNG wire#powerrail
      Contact( "LaserComm".Instance[#iInstance_Index].Scanner.Reset )
   END_RUNG wire#w1
   RUNG wire#w1
      { S7_GenerateENO := "TRUE" } Move(in := 0, out1 => #sCTU.CV)
   END_RUNG
   // the same network as SCL:
   // ENO of a box is taken as its EN; it also drops when the box reports an error
   #_w1 := (#sNo_Faults_Active AND (#sStep = 40)) OR "LaserComm".Instance[#iInstance_Index].Scanner.Reset;
   #_w2 := (#sNo_Faults_Active AND (#sStep = 40)) OR "LaserComm".Instance[#iInstance_Index].Scanner.Reset;
   IF #_w2 THEN
       #sStep := 0;
       #sCounter_Done := FALSE;
   END_IF;
   IF #_w1 THEN #sCTU.CV := 0; END_IF;
END_REGION
END_FUNCTION_BLOCK

FUNCTION_BLOCK "Call"   // FB1, LAD
{ S7_Optimized_Access := 'TRUE' }
VERSION : 0.1
// stored: AutoNumber true, IsIECCheckEnabled false, IsRetainMemResEnabled false, MemoryReserve 100, SetENOAutomatically false, UDAEnableTagReadback false
   VAR
      LaserComm_API_Instance { S7_SetPoint := 'True'} : Array[0..1] of "LaserComm_API";
      Dummy_Cereal_Number { S7_SetPoint := 'True'} : Array[1..32] of Char;
      Dummy_Part_Type { S7_SetPoint := 'True'} : Array[1..18] of Char;
   END_VAR
BEGIN

REGION Network 2: IPG and OPC FB Calls
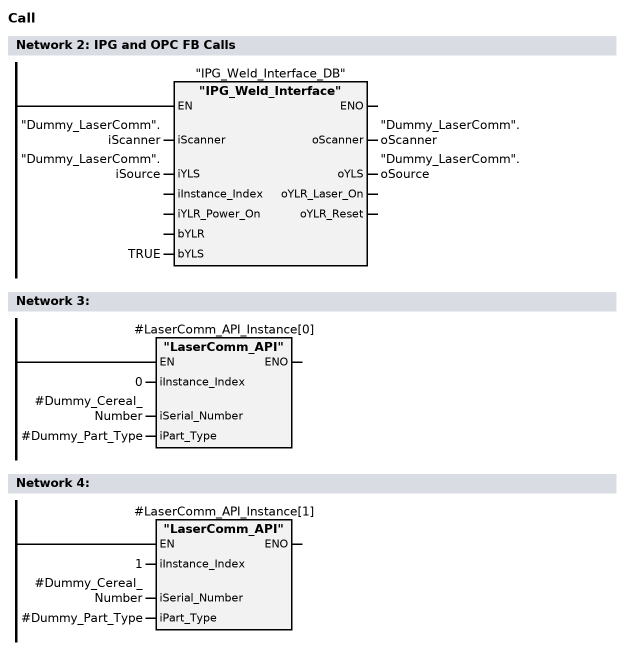
   RUNG wire#powerrail
      "IPG_Weld_Interface_DB"(iScanner := "Dummy_LaserComm".iScanner, iYLS := "Dummy_LaserComm".iSource, iInstance_Index :=, iYLR_Power_On :=, bYLR :=, bYLS := TRUE, oScanner => "Dummy_LaserComm".oScanner, oYLS => "Dummy_LaserComm".oSource, oYLR_Laser_On =>, oYLR_Reset =>)
   END_RUNG
   // the same network as SCL:
   "IPG_Weld_Interface_DB"(iScanner := "Dummy_LaserComm".iScanner,   // "IPG_Weld_Interface"
                           iYLS := "Dummy_LaserComm".iSource,
                           bYLS := TRUE,
                           oScanner => "Dummy_LaserComm".oScanner,
                           oYLS => "Dummy_LaserComm".oSource);
END_REGION

REGION Network 3
   RUNG wire#powerrail
      #LaserComm_API_Instance[0](iInstance_Index := 0, iSerial_Number := #Dummy_Cereal_Number, iPart_Type := #Dummy_Part_Type)
   END_RUNG
   // the same network as SCL:
   #LaserComm_API_Instance[0](iInstance_Index := 0,   // "LaserComm_API"
                           iSerial_Number := #Dummy_Cereal_Number,
                           iPart_Type := #Dummy_Part_Type);
END_REGION

REGION Network 4
   RUNG wire#powerrail
      #LaserComm_API_Instance[1](iInstance_Index := 1, iSerial_Number := #Dummy_Cereal_Number, iPart_Type := #Dummy_Part_Type)
   END_RUNG
   // the same network as SCL:
   #LaserComm_API_Instance[1](iInstance_Index := 1,   // "LaserComm_API"
                           iSerial_Number := #Dummy_Cereal_Number,
                           iPart_Type := #Dummy_Part_Type);
END_REGION
END_FUNCTION_BLOCK

FUNCTION_BLOCK "IPG_Weld_Interface"   // FB304, LAD
TITLE = IPG Communication Handling / IPG Weld Interface
{ S7_Optimized_Access := 'FALSE' }
VERSION : 1.0
// stored: AutoNumber true, IsIECCheckEnabled false, SetENOAutomatically false, UDAEnableTagReadback false
   VAR_INPUT
      iScanner : "Scanner_Inputs";
      iYLS : "YLS_Inputs";
      iInstance_Index : Int;
      iYLR_Power_On : Bool;
      bYLR : Bool;
      bYLS : Bool;
   END_VAR
   VAR_OUTPUT
      oScanner : "Scanner_Outputs";
      oYLS : "YLS_Outputs";
      oYLR_Laser_On : Bool;
      oYLR_Reset : Bool;
   END_VAR
   VAR DB_SPECIFIC
      sStep : Int;
      sLast_Step : Int;
      sScanner_Idle : Bool;
      sScanner_Active : Bool;
      sScanner_Error : Bool;
      sScanner_Waiting_Enable : Bool;
      sScanner_Waiting_Strobe : Bool;
      sScanner_Waiting_Start : Bool;
      tJob_Start_ONS { ExternalAccessible := 'False'; ExternalVisible := 'False'; ExternalWritable := 'False'} : Bool;
      tJob_Stop_ONS { ExternalAccessible := 'False'; ExternalVisible := 'False'; ExternalWritable := 'False'} : Bool;
      siScanner_Job : Byte;
      siScanner_Group : Byte;
      soScanner_Job : Byte;
      soScanner_Group : Byte;
      sVersion { S7_SetPoint := 'True'} : Real;
      sStepTimeout : IEC_TIMER;
      sReset_Timer { S7_SetPoint := 'True'} : IEC_TIMER;
      sLog : Array[0..50] of Struct
         Load_Start_Time : Date_And_Time;
         Load_Stop_Time : Date_And_Time;
         Fire_Start_Time : Date_And_Time;
         Fire_Stop_Time : Date_And_Time;
         Job_ID : Byte;
         Group_ID : Byte;
      END_STRUCT;
      sBlankLog : Struct
         Load_Start_Time : Date_And_Time;
         Load_Stop_Time : Date_And_Time;
         Fire_Start_Time : Date_And_Time;
         Fire_Stop_Time : Date_And_Time;
         Job_ID : Byte;
         Group_ID : Byte;
      END_STRUCT;
   END_VAR
   VAR_TEMP
      tLasRes : Bool;
      tStep_Changed_ONS : Bool;
      tPointer : Int;
      tStart_Load_Int : Int;
      tStop_Load_Int : Int;
      tStart_Fire_Int : Int;
      tStop_Fire_Int : Int;
   END_VAR
   VAR_TEMP   // added for the SCL form of the ladder/FBD networks
      _w1 : Bool;
      _w2 : Bool;
   END_VAR
BEGIN

REGION Network 1: Version
   // V1.1
   // Mapped all Scanner and YLS Inputs and Outputs
   // V1.2
   // Added YLR Faults and Interface (need to add condition for Power On of YLR)
   // V2
   // Laser Comm DB Reorder, remove redunudant logic
   // Added Job and Group Log
   // Removed Guide Beam On Fault. Soace reserved.
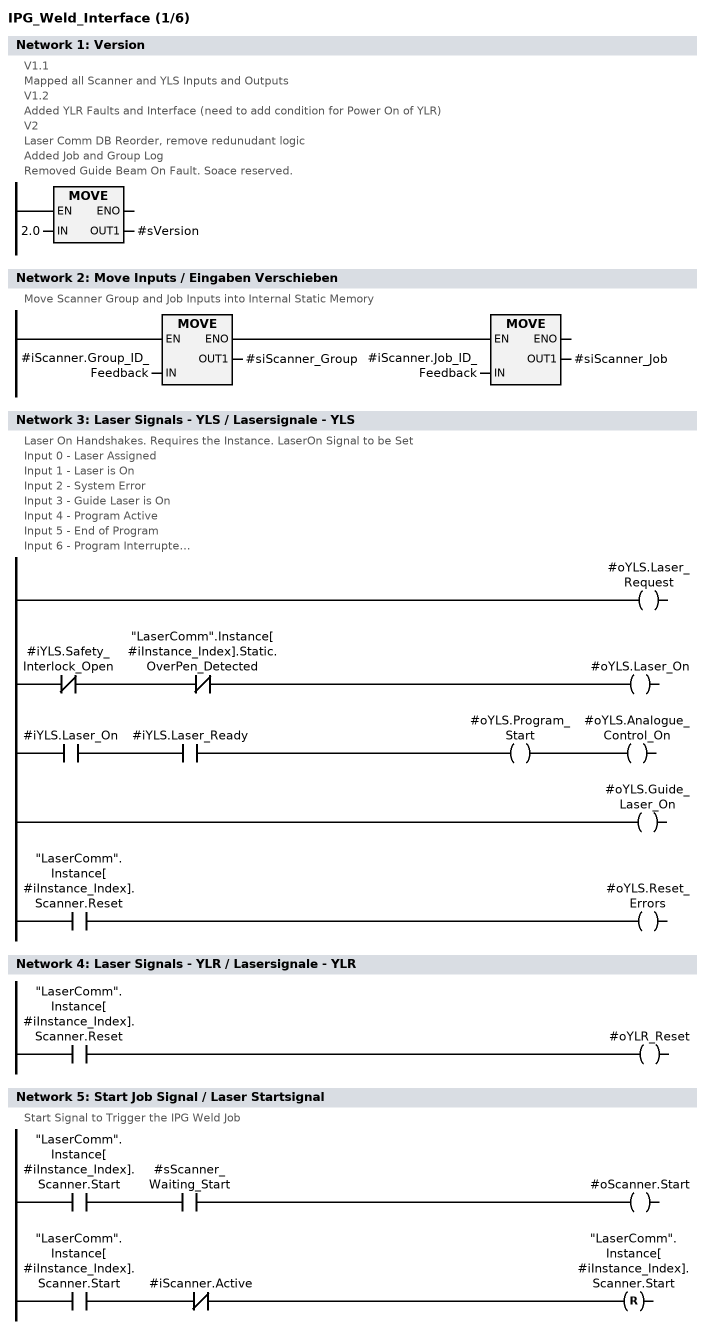
   RUNG wire#powerrail
      Move(in := 2.0, out1 => #sVersion)
   END_RUNG
   // the same network as SCL:
   #sVersion := 2.0;
END_REGION

REGION Network 2: Move Inputs / Eingaben Verschieben
   // Move Scanner Group and Job Inputs into Internal Static Memory
   RUNG wire#powerrail
      Move(in := #iScanner.Group_ID_Feedback, out1 => #siScanner_Group)
      Move(in := #iScanner.Job_ID_Feedback, out1 => #siScanner_Job)
   END_RUNG
   // the same network as SCL:
   #siScanner_Group := #iScanner.Group_ID_Feedback;
   #siScanner_Job := #iScanner.Job_ID_Feedback;
END_REGION

REGION Network 3: Laser Signals - YLS / Lasersignale - YLS
   // Laser On Handshakes. Requires the Instance. LaserOn Signal to be Set
   // Input 0 - Laser Assigned
   // Input 1 - Laser is On
   // Input 2 - System Error
   // Input 3 - Guide Laser is On
   // Input 4 - Program Active
   // Input 5 - End of Program
   // Input 6 - Program Interrupted
   // Input 7 - Analogue Control is On
   // Input 8 - System Warning
   // Input 9 - Laser Ready
   // Input 10 - Emission On
   // 
   // Output 0 - Laser Request (should always be On)
   // Output 1 - Laser On
   // Output 2 - Reset Errors
   // Output 3 - Guide Laser On
   // Output 4 - Program Start
   // Output 5 - Program Stop
   // Output 6 - Reserved
   // Output 7 - Analogue Control On
   RUNG wire#powerrail
      Coil( #oYLS.Laser_Request )
   END_RUNG
   RUNG wire#powerrail
      I_Contact( #iYLS.Safety_Interlock_Open )
      I_Contact( "LaserComm".Instance[#iInstance_Index].Static.OverPen_Detected )
      Coil( #oYLS.Laser_On )
   END_RUNG
   RUNG wire#powerrail
      Contact( #iYLS.Laser_On )
      Contact( #iYLS.Laser_Ready )
      Coil( #oYLS.Program_Start )
      Coil( #oYLS.Analogue_Control_On )
   END_RUNG
   RUNG wire#powerrail
      Coil( #oYLS.Guide_Laser_On )
   END_RUNG
   RUNG wire#powerrail
      Contact( "LaserComm".Instance[#iInstance_Index].Scanner.Reset )
      Coil( #oYLS.Reset_Errors )
   END_RUNG
   // the same network as SCL:
   #oYLS.Laser_Request := TRUE;
   #oYLS.Laser_On := NOT #iYLS.Safety_Interlock_Open AND NOT "LaserComm".Instance[#iInstance_Index].Static.OverPen_Detected;
   #oYLS.Program_Start := #iYLS.Laser_On AND #iYLS.Laser_Ready;
   #oYLS.Analogue_Control_On := #oYLS.Program_Start;
   #oYLS.Guide_Laser_On := TRUE;
   #oYLS.Reset_Errors := "LaserComm".Instance[#iInstance_Index].Scanner.Reset;
END_REGION

REGION Network 4: Laser Signals - YLR / Lasersignale - YLR
   RUNG wire#powerrail
      Contact( "LaserComm".Instance[#iInstance_Index].Scanner.Reset )
      Coil( #oYLR_Reset )
   END_RUNG
   // the same network as SCL:
   #oYLR_Reset := "LaserComm".Instance[#iInstance_Index].Scanner.Reset;
END_REGION

REGION Network 5: Start Job Signal / Laser Startsignal
   // Start Signal to Trigger the IPG Weld Job
   RUNG wire#powerrail
      Contact( "LaserComm".Instance[#iInstance_Index].Scanner.Start )
      Contact( #sScanner_Waiting_Start )
      Coil( #oScanner.Start )
   END_RUNG
   RUNG wire#powerrail
      Contact( "LaserComm".Instance[#iInstance_Index].Scanner.Start )
      I_Contact( #iScanner.Active )
      R_Coil( "LaserComm".Instance[#iInstance_Index].Scanner.Start )
   END_RUNG
   // the same network as SCL:
   #oScanner.Start := "LaserComm".Instance[#iInstance_Index].Scanner.Start AND #sScanner_Waiting_Start;
   IF "LaserComm".Instance[#iInstance_Index].Scanner.Start AND NOT #iScanner.Active THEN
       "LaserComm".Instance[#iInstance_Index].Scanner.Start := FALSE;
   END_IF;
END_REGION

REGION Network 6: Log Fire Time Handling
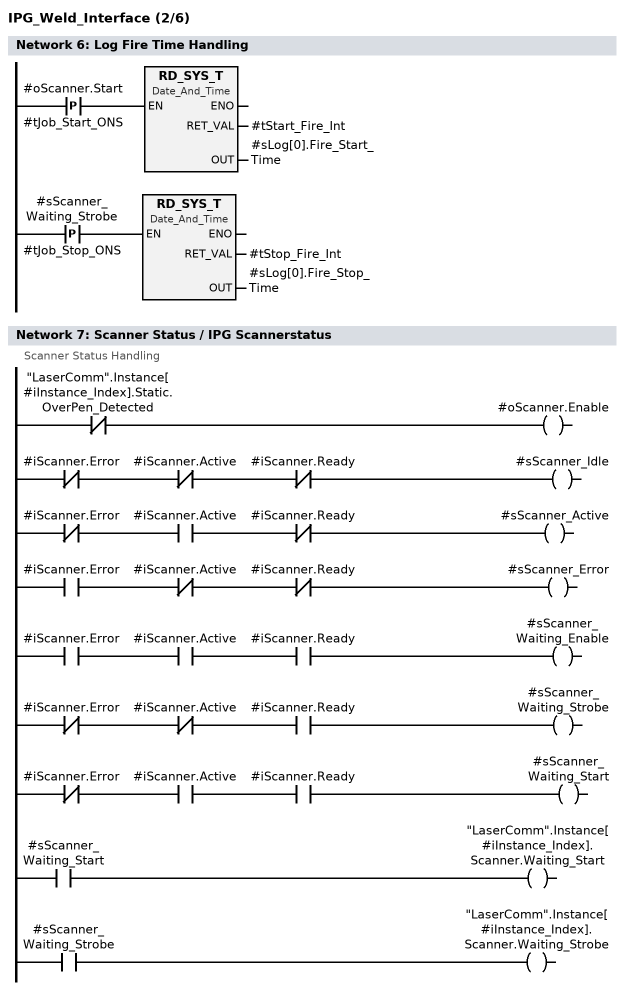
   RUNG wire#powerrail
      P_Contact(operand := #oScanner.Start, bit := #tJob_Start_ONS)
      { S7_Templates := "date_type := Date_And_Time" } RD_SYS_T(RET_VAL => #tStart_Fire_Int, OUT => #sLog[0].Fire_Start_Time)
   END_RUNG
   RUNG wire#powerrail
      P_Contact(operand := #sScanner_Waiting_Strobe, bit := #tJob_Stop_ONS)
      { S7_Templates := "date_type := Date_And_Time" } RD_SYS_T(RET_VAL => #tStop_Fire_Int, OUT => #sLog[0].Fire_Stop_Time)
   END_RUNG
   // the same network as SCL:
   #_w1 := #oScanner.Start AND NOT #tJob_Start_ONS;   // rising edge of #oScanner.Start
   #tJob_Start_ONS := #oScanner.Start;
   IF #_w1 THEN #tStart_Fire_Int := RD_SYS_T(OUT => #sLog[0].Fire_Start_Time); END_IF;
   #_w2 := #sScanner_Waiting_Strobe AND NOT #tJob_Stop_ONS;   // rising edge of #sScanner_Waiting_Strobe
   #tJob_Stop_ONS := #sScanner_Waiting_Strobe;
   IF #_w2 THEN #tStop_Fire_Int := RD_SYS_T(OUT => #sLog[0].Fire_Stop_Time); END_IF;
END_REGION

REGION Network 7: Scanner Status / IPG Scannerstatus
   // Scanner Status Handling
   RUNG wire#powerrail
      I_Contact( "LaserComm".Instance[#iInstance_Index].Static.OverPen_Detected )
      Coil( #oScanner.Enable )
   END_RUNG
   RUNG wire#powerrail
      I_Contact( #iScanner.Error )
      I_Contact( #iScanner.Active )
      I_Contact( #iScanner.Ready )
      Coil( #sScanner_Idle )
   END_RUNG
   RUNG wire#powerrail
      I_Contact( #iScanner.Error )
      Contact( #iScanner.Active )
      I_Contact( #iScanner.Ready )
      Coil( #sScanner_Active )
   END_RUNG
   RUNG wire#powerrail
      Contact( #iScanner.Error )
      I_Contact( #iScanner.Active )
      I_Contact( #iScanner.Ready )
      Coil( #sScanner_Error )
   END_RUNG
   RUNG wire#powerrail
      Contact( #iScanner.Error )
      Contact( #iScanner.Active )
      Contact( #iScanner.Ready )
      Coil( #sScanner_Waiting_Enable )
   END_RUNG
   RUNG wire#powerrail
      I_Contact( #iScanner.Error )
      I_Contact( #iScanner.Active )
      Contact( #iScanner.Ready )
      Coil( #sScanner_Waiting_Strobe )
   END_RUNG
   RUNG wire#powerrail
      I_Contact( #iScanner.Error )
      Contact( #iScanner.Active )
      Contact( #iScanner.Ready )
      Coil( #sScanner_Waiting_Start )
   END_RUNG
   RUNG wire#powerrail
      Contact( #sScanner_Waiting_Start )
      Coil( "LaserComm".Instance[#iInstance_Index].Scanner.Waiting_Start )
   END_RUNG
   RUNG wire#powerrail
      Contact( #sScanner_Waiting_Strobe )
      Coil( "LaserComm".Instance[#iInstance_Index].Scanner.Waiting_Strobe )
   END_RUNG
   // the same network as SCL:
   #oScanner.Enable := NOT "LaserComm".Instance[#iInstance_Index].Static.OverPen_Detected;
   #sScanner_Idle := NOT #iScanner.Error AND NOT #iScanner.Active AND NOT #iScanner.Ready;
   #sScanner_Active := NOT #iScanner.Error AND #iScanner.Active AND NOT #iScanner.Ready;
   #sScanner_Error := #iScanner.Error AND NOT #iScanner.Active AND NOT #iScanner.Ready;
   #sScanner_Waiting_Enable := #iScanner.Error AND #iScanner.Active AND #iScanner.Ready;
   #sScanner_Waiting_Strobe := NOT #iScanner.Error AND NOT #iScanner.Active AND #iScanner.Ready;
   #sScanner_Waiting_Start := NOT #iScanner.Error AND #iScanner.Active AND #iScanner.Ready;
   "LaserComm".Instance[#iInstance_Index].Scanner.Waiting_Start := #sScanner_Waiting_Start;
   "LaserComm".Instance[#iInstance_Index].Scanner.Waiting_Strobe := #sScanner_Waiting_Strobe;
END_REGION

REGION Network 8: Step 0 / Schritt 0
   // Initial Step. Wait for Scanner Ready to Begin with Job and Group Not 0. / Job und Gruppen ID Laden
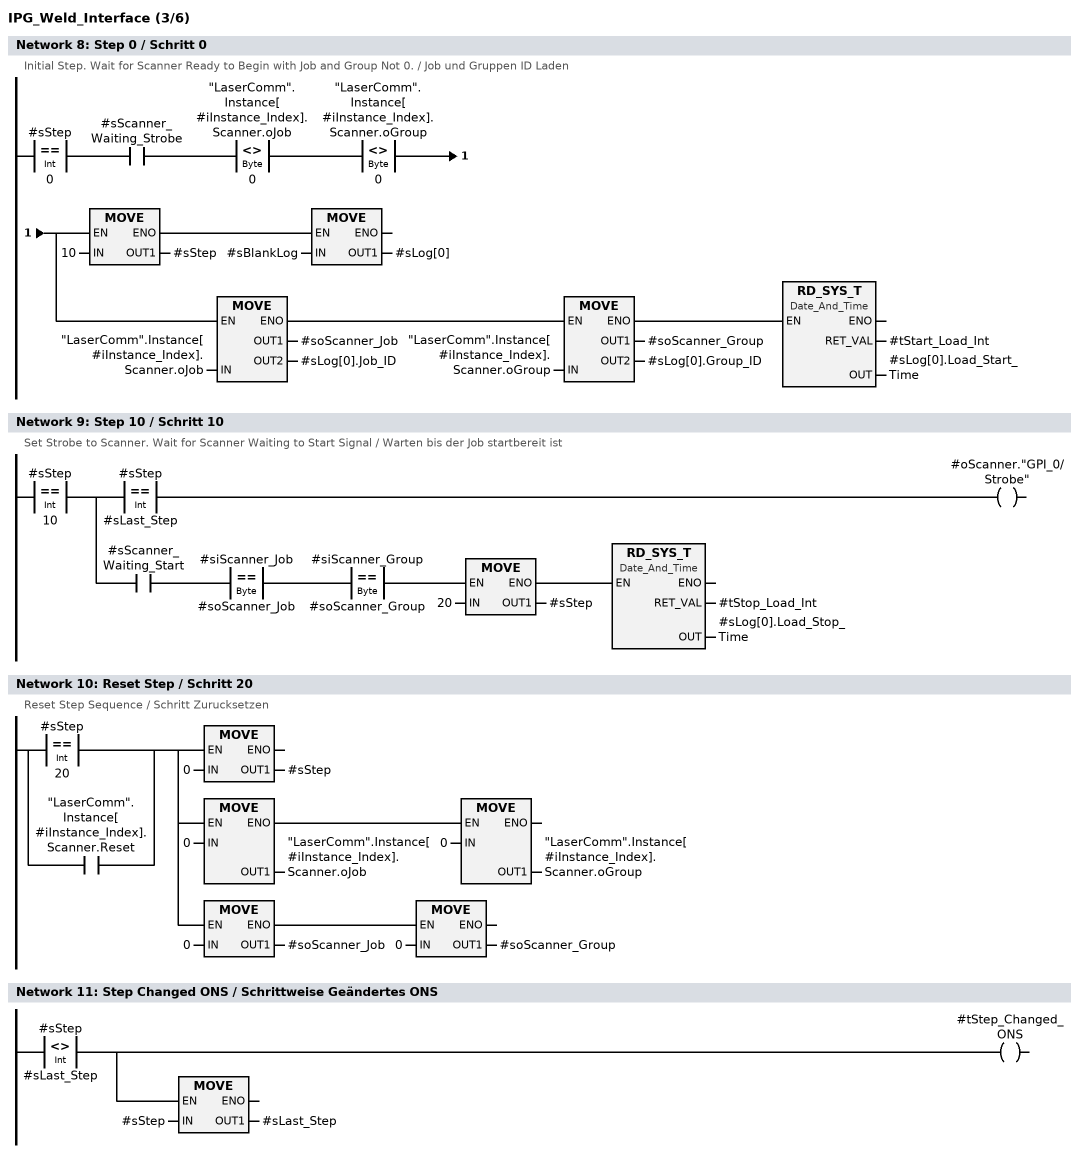
   RUNG wire#powerrail
      { S7_Templates := "SrcType := Int" } EQ_Contact(in1 := #sStep, in2 := 0)
      Contact( #sScanner_Waiting_Strobe )
      { S7_Templates := "SrcType := Byte" } NE_Contact(in1 := "LaserComm".Instance[#iInstance_Index].Scanner.oJob, in2 := 0)
      { S7_Templates := "SrcType := Byte" } NE_Contact(in1 := "LaserComm".Instance[#iInstance_Index].Scanner.oGroup, in2 := 0)
      wire#w1
      Move(in := 10, out1 => #sStep)
      Move(in := #sBlankLog, out1 => #sLog[0])
   END_RUNG
   RUNG wire#w1
      Move(in := "LaserComm".Instance[#iInstance_Index].Scanner.oJob, out1 => #soScanner_Job, out2 => #sLog[0].Job_ID)
      Move(in := "LaserComm".Instance[#iInstance_Index].Scanner.oGroup, out1 => #soScanner_Group, out2 => #sLog[0].Group_ID)
      { S7_Templates := "date_type := Date_And_Time" } RD_SYS_T(RET_VAL => #tStart_Load_Int, OUT => #sLog[0].Load_Start_Time)
   END_RUNG
   // the same network as SCL:
   #_w1 := (#sStep = 0) AND #sScanner_Waiting_Strobe AND ("LaserComm".Instance[#iInstance_Index].Scanner.oJob <> 0) AND ("LaserComm".Instance[#iInstance_Index].Scanner.oGroup <> 0);
   #_w2 := (#sStep = 0) AND #sScanner_Waiting_Strobe AND ("LaserComm".Instance[#iInstance_Index].Scanner.oJob <> 0) AND ("LaserComm".Instance[#iInstance_Index].Scanner.oGroup <> 0);
   IF #_w2 THEN
       #sStep := 10;
       #sLog[0] := #sBlankLog;
   END_IF;
   IF #_w1 THEN
       #soScanner_Job := "LaserComm".Instance[#iInstance_Index].Scanner.oJob;
       #sLog[0].Job_ID := "LaserComm".Instance[#iInstance_Index].Scanner.oJob;
       #soScanner_Group := "LaserComm".Instance[#iInstance_Index].Scanner.oGroup;
       #sLog[0].Group_ID := "LaserComm".Instance[#iInstance_Index].Scanner.oGroup;
       #tStart_Load_Int := RD_SYS_T(OUT => #sLog[0].Load_Start_Time);
   END_IF;
END_REGION

REGION Network 9: Step 10 / Schritt 10
   // Set Strobe to Scanner. Wait for Scanner Waiting to Start Signal / Warten bis der Job startbereit ist
   RUNG wire#powerrail
      { S7_Templates := "SrcType := Int" } EQ_Contact(in1 := #sStep, in2 := 10)
      wire#w1
      { S7_Templates := "SrcType := Int" } EQ_Contact(in1 := #sStep, in2 := #sLast_Step)
      Coil( #oScanner."GPI_0/Strobe" )
   END_RUNG
   RUNG wire#w1
      Contact( #sScanner_Waiting_Start )
      { S7_Templates := "SrcType := Byte" } EQ_Contact(in1 := #siScanner_Job, in2 := #soScanner_Job)
      { S7_Templates := "SrcType := Byte" } EQ_Contact(in1 := #siScanner_Group, in2 := #soScanner_Group)
      Move(in := 20, out1 => #sStep)
      { S7_Templates := "date_type := Date_And_Time" } RD_SYS_T(RET_VAL => #tStop_Load_Int, OUT => #sLog[0].Load_Stop_Time)
   END_RUNG
   // the same network as SCL:
   #_w1 := #sStep = 10;
   #oScanner."GPI_0/Strobe" := #_w1 AND (#sStep = #sLast_Step);
   IF #_w1 AND #sScanner_Waiting_Start AND (#siScanner_Job = #soScanner_Job) AND (#siScanner_Group = #soScanner_Group) THEN
       #sStep := 20;
       #tStop_Load_Int := RD_SYS_T(OUT => #sLog[0].Load_Stop_Time);
   END_IF;
END_REGION

REGION Network 10: Reset Step / Schritt 20
   // Reset Step Sequence / Schritt Zurucksetzen
   RUNG wire#powerrail
      { S7_Templates := "SrcType := Int" } EQ_Contact(in1 := #sStep, in2 := 20)
      wire#w1
      Move(in := 0, out1 => #sStep)
   END_RUNG
   RUNG wire#powerrail
      Contact( "LaserComm".Instance[#iInstance_Index].Scanner.Reset )
   END_RUNG wire#w1
   RUNG wire#w1
      Move(in := 0, out1 => "LaserComm".Instance[#iInstance_Index].Scanner.oJob)
      Move(in := 0, out1 => "LaserComm".Instance[#iInstance_Index].Scanner.oGroup)
   END_RUNG
   RUNG wire#w1
      Move(in := 0, out1 => #soScanner_Job)
      Move(in := 0, out1 => #soScanner_Group)
   END_RUNG
   // the same network as SCL:
   #_w1 := (#sStep = 20) OR "LaserComm".Instance[#iInstance_Index].Scanner.Reset;
   IF #_w1 THEN
       #sStep := 0;
       "LaserComm".Instance[#iInstance_Index].Scanner.oJob := 0;
       "LaserComm".Instance[#iInstance_Index].Scanner.oGroup := 0;
       #soScanner_Job := 0;
       #soScanner_Group := 0;
   END_IF;
END_REGION

REGION Network 11: Step Changed ONS / Schrittweise Geändertes ONS
   RUNG wire#powerrail
      { S7_Templates := "SrcType := Int" } NE_Contact(in1 := #sStep, in2 := #sLast_Step)
      wire#w1
      Coil( #tStep_Changed_ONS )
   END_RUNG
   RUNG wire#w1
      { S7_GenerateENO := "TRUE" } Move(in := #sStep, out1 => #sLast_Step)
   END_RUNG
   // the same network as SCL:
   #tStep_Changed_ONS := #sStep <> #sLast_Step;
   IF #tStep_Changed_ONS THEN #sLast_Step := #sStep; END_IF;
END_REGION

REGION Network 12: Reset Flag / Reset Flag Entrigein
   // Clear Reset Flag - Timer Required as Laser Source requires a duration pulse to reset
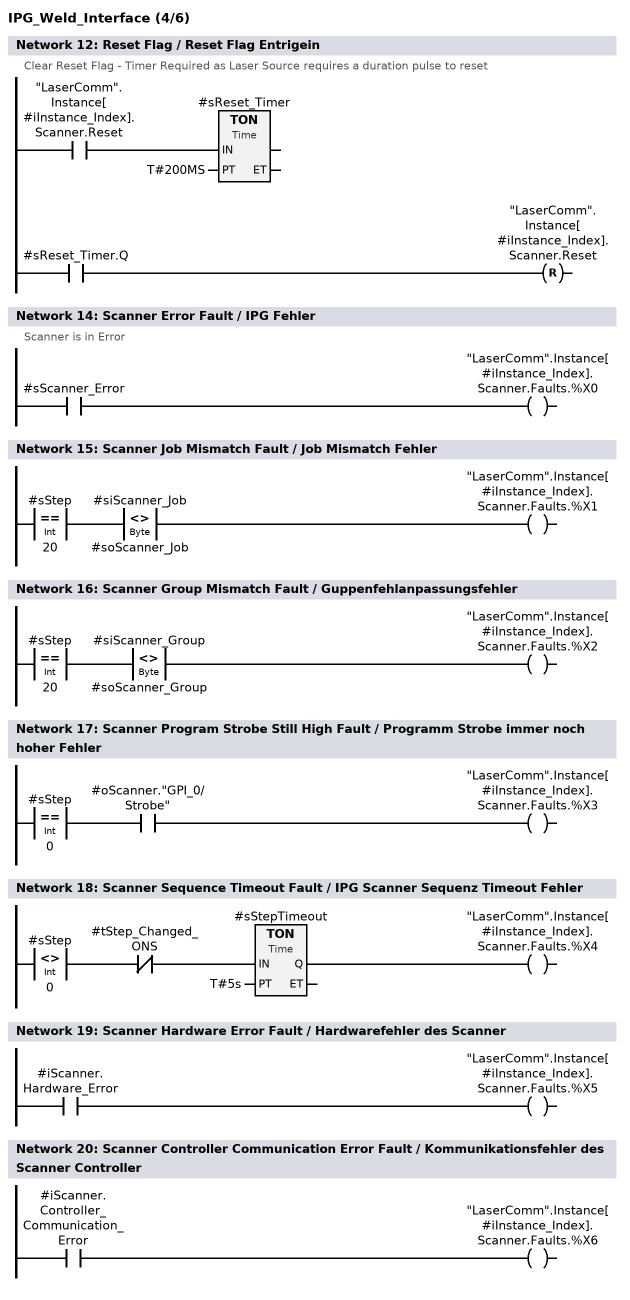
   RUNG wire#powerrail
      Contact( "LaserComm".Instance[#iInstance_Index].Scanner.Reset )
      { S7_Templates := "time_type := Time" } #sReset_Timer.TON(pt := T#200MS, et =>)
   END_RUNG
   RUNG wire#powerrail
      Contact( #sReset_Timer.Q )
      R_Coil( "LaserComm".Instance[#iInstance_Index].Scanner.Reset )
   END_RUNG
   // the same network as SCL:
   #sReset_Timer.TON(IN := "LaserComm".Instance[#iInstance_Index].Scanner.Reset, PT := T#200MS);
   IF #sReset_Timer.Q THEN "LaserComm".Instance[#iInstance_Index].Scanner.Reset := FALSE; END_IF;
END_REGION

REGION Network 13 (SCL): Job Log Handler
   // Records when the last job and group was loaded and fired
   // Job Log Handler

   IF #sLog[0].Job_ID <> 0 AND #sLog[0].Group_ID <> 0 AND #sLog[0].Fire_Stop_Time <> DT#1990-01-01-00:00:00 THEN
       FOR #tPointer := 49 TO 0 BY -1 DO
           #sLog[#tPointer + 1] := #sLog[#tPointer];
       END_FOR;

       #sLog[0] := #sBlankLog;

   END_IF;
END_REGION

REGION Network 14: Scanner Error Fault / IPG Fehler
   // Scanner is in Error
   RUNG wire#powerrail
      Contact( #sScanner_Error )
      Coil( "LaserComm".Instance[#iInstance_Index].Scanner.Faults.%X0 )
   END_RUNG
   // the same network as SCL:
   "LaserComm".Instance[#iInstance_Index].Scanner.Faults.%X0 := #sScanner_Error;
END_REGION

REGION Network 15: Scanner Job Mismatch Fault / Job Mismatch Fehler
   RUNG wire#powerrail
      { S7_Templates := "SrcType := Int" } EQ_Contact(in1 := #sStep, in2 := 20)
      { S7_Templates := "SrcType := Byte" } NE_Contact(in1 := #siScanner_Job, in2 := #soScanner_Job)
      Coil( "LaserComm".Instance[#iInstance_Index].Scanner.Faults.%X1 )
   END_RUNG
   // the same network as SCL:
   "LaserComm".Instance[#iInstance_Index].Scanner.Faults.%X1 := (#sStep = 20) AND (#siScanner_Job <> #soScanner_Job);
END_REGION

REGION Network 16: Scanner Group Mismatch Fault / Guppenfehlanpassungsfehler
   RUNG wire#powerrail
      { S7_Templates := "SrcType := Int" } EQ_Contact(in1 := #sStep, in2 := 20)
      { S7_Templates := "SrcType := Byte" } NE_Contact(in1 := #siScanner_Group, in2 := #soScanner_Group)
      Coil( "LaserComm".Instance[#iInstance_Index].Scanner.Faults.%X2 )
   END_RUNG
   // the same network as SCL:
   "LaserComm".Instance[#iInstance_Index].Scanner.Faults.%X2 := (#sStep = 20) AND (#siScanner_Group <> #soScanner_Group);
END_REGION

REGION Network 17: Scanner Program Strobe Still High Fault / Programm Strobe immer noch hoher Fehler
   RUNG wire#powerrail
      { S7_Templates := "SrcType := Int" } EQ_Contact(in1 := #sStep, in2 := 0)
      Contact( #oScanner."GPI_0/Strobe" )
      Coil( "LaserComm".Instance[#iInstance_Index].Scanner.Faults.%X3 )
   END_RUNG
   // the same network as SCL:
   "LaserComm".Instance[#iInstance_Index].Scanner.Faults.%X3 := (#sStep = 0) AND #oScanner."GPI_0/Strobe";
END_REGION

REGION Network 18: Scanner Sequence Timeout Fault / IPG Scanner Sequenz Timeout Fehler
   RUNG wire#powerrail
      { S7_Templates := "SrcType := Int" } NE_Contact(in1 := #sStep, in2 := 0)
      I_Contact( #tStep_Changed_ONS )
      { S7_Templates := "time_type := Time" } #sStepTimeout.TON(pt := T#5s, et =>)
      Coil( "LaserComm".Instance[#iInstance_Index].Scanner.Faults.%X4 )
   END_RUNG
   // the same network as SCL:
   #sStepTimeout.TON(IN := (#sStep <> 0) AND NOT #tStep_Changed_ONS, PT := T#5s);
   "LaserComm".Instance[#iInstance_Index].Scanner.Faults.%X4 := #sStepTimeout.Q;
END_REGION

REGION Network 19: Scanner Hardware Error Fault / Hardwarefehler des Scanner
   RUNG wire#powerrail
      Contact( #iScanner.Hardware_Error )
      Coil( "LaserComm".Instance[#iInstance_Index].Scanner.Faults.%X5 )
   END_RUNG
   // the same network as SCL:
   "LaserComm".Instance[#iInstance_Index].Scanner.Faults.%X5 := #iScanner.Hardware_Error;
END_REGION

REGION Network 20: Scanner Controller Communication Error Fault / Kommunikationsfehler des Scanner Controller
   RUNG wire#powerrail
      Contact( #iScanner.Controller_Communication_Error )
      Coil( "LaserComm".Instance[#iInstance_Index].Scanner.Faults.%X6 )
   END_RUNG
   // the same network as SCL:
   "LaserComm".Instance[#iInstance_Index].Scanner.Faults.%X6 := #iScanner.Controller_Communication_Error;
END_REGION

REGION Network 21: Scanner Head Communication Error Fault / Fehler bei derKommunikation mit dem Scannerkopf
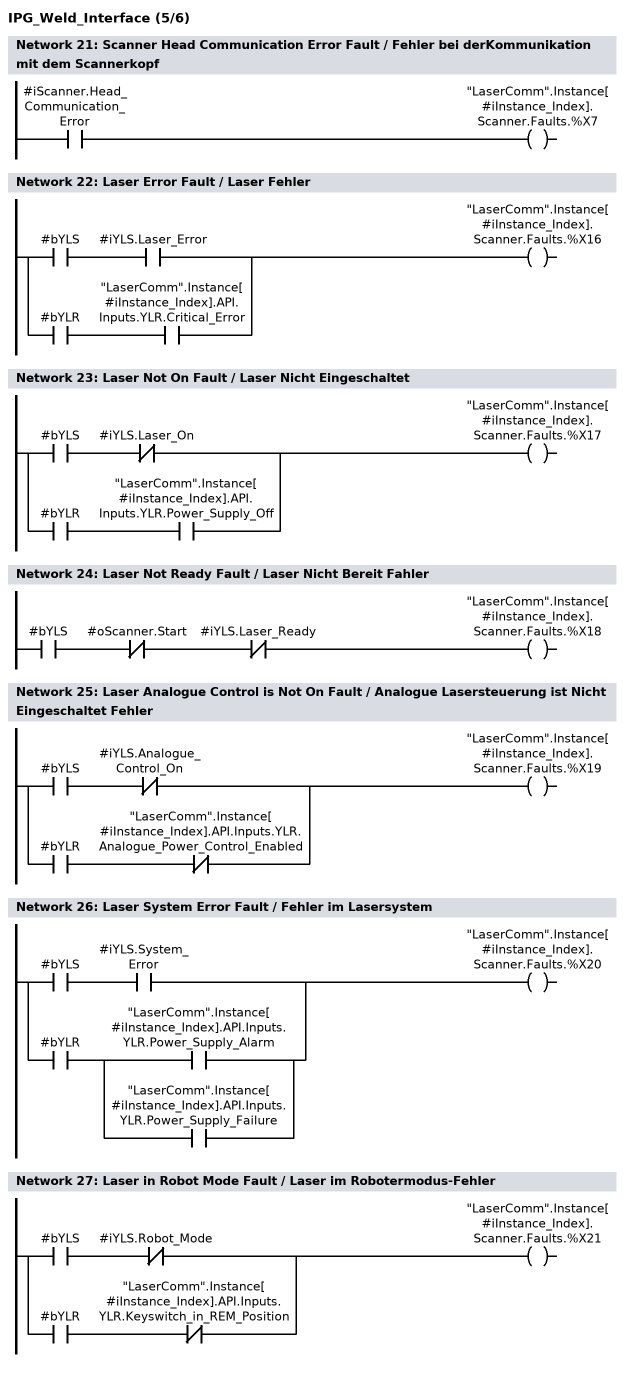
   RUNG wire#powerrail
      Contact( #iScanner.Head_Communication_Error )
      Coil( "LaserComm".Instance[#iInstance_Index].Scanner.Faults.%X7 )
   END_RUNG
   // the same network as SCL:
   "LaserComm".Instance[#iInstance_Index].Scanner.Faults.%X7 := #iScanner.Head_Communication_Error;
END_REGION

REGION Network 22: Laser Error Fault / Laser Fehler
   RUNG wire#powerrail
      Contact( #bYLS )
      Contact( #iYLS.Laser_Error )
      wire#w1
      Coil( "LaserComm".Instance[#iInstance_Index].Scanner.Faults.%X16 )
   END_RUNG
   RUNG wire#powerrail
      Contact( #bYLR )
      Contact( "LaserComm".Instance[#iInstance_Index].API.Inputs.YLR.Critical_Error )
   END_RUNG wire#w1
   // the same network as SCL:
   "LaserComm".Instance[#iInstance_Index].Scanner.Faults.%X16 := (#bYLS AND #iYLS.Laser_Error) OR (#bYLR AND "LaserComm".Instance[#iInstance_Index].API.Inputs.YLR.Critical_Error);
END_REGION

REGION Network 23: Laser Not On Fault / Laser Nicht Eingeschaltet
   RUNG wire#powerrail
      Contact( #bYLS )
      I_Contact( #iYLS.Laser_On )
      wire#w1
      Coil( "LaserComm".Instance[#iInstance_Index].Scanner.Faults.%X17 )
   END_RUNG
   RUNG wire#powerrail
      Contact( #bYLR )
      Contact( "LaserComm".Instance[#iInstance_Index].API.Inputs.YLR.Power_Supply_Off )
   END_RUNG wire#w1
   // the same network as SCL:
   "LaserComm".Instance[#iInstance_Index].Scanner.Faults.%X17 := (#bYLS AND NOT #iYLS.Laser_On) OR (#bYLR AND "LaserComm".Instance[#iInstance_Index].API.Inputs.YLR.Power_Supply_Off);
END_REGION

REGION Network 24: Laser Not Ready Fault / Laser Nicht Bereit Fahler
   RUNG wire#powerrail
      Contact( #bYLS )
      I_Contact( #oScanner.Start )
      I_Contact( #iYLS.Laser_Ready )
      Coil( "LaserComm".Instance[#iInstance_Index].Scanner.Faults.%X18 )
   END_RUNG
   // the same network as SCL:
   "LaserComm".Instance[#iInstance_Index].Scanner.Faults.%X18 := #bYLS AND NOT #oScanner.Start AND NOT #iYLS.Laser_Ready;
END_REGION

REGION Network 25: Laser Analogue Control is Not On Fault / Analogue Lasersteuerung ist Nicht Eingeschaltet Fehler
   RUNG wire#powerrail
      Contact( #bYLS )
      I_Contact( #iYLS.Analogue_Control_On )
      wire#w1
      Coil( "LaserComm".Instance[#iInstance_Index].Scanner.Faults.%X19 )
   END_RUNG
   RUNG wire#powerrail
      Contact( #bYLR )
      I_Contact( "LaserComm".Instance[#iInstance_Index].API.Inputs.YLR.Analogue_Power_Control_Enabled )
   END_RUNG wire#w1
   // the same network as SCL:
   "LaserComm".Instance[#iInstance_Index].Scanner.Faults.%X19 := (#bYLS AND NOT #iYLS.Analogue_Control_On) OR (#bYLR AND NOT "LaserComm".Instance[#iInstance_Index].API.Inputs.YLR.Analogue_Power_Control_Enabled);
END_REGION

REGION Network 26: Laser System Error Fault / Fehler im Lasersystem
   RUNG wire#powerrail
      Contact( #bYLS )
      Contact( #iYLS.System_Error )
      wire#w1
      Coil( "LaserComm".Instance[#iInstance_Index].Scanner.Faults.%X20 )
   END_RUNG
   RUNG wire#powerrail
      Contact( #bYLR )
      wire#w2
      Contact( "LaserComm".Instance[#iInstance_Index].API.Inputs.YLR.Power_Supply_Alarm )
   END_RUNG wire#w1
   RUNG wire#w2
      Contact( "LaserComm".Instance[#iInstance_Index].API.Inputs.YLR.Power_Supply_Failure )
   END_RUNG wire#w1
   // the same network as SCL:
   "LaserComm".Instance[#iInstance_Index].Scanner.Faults.%X20 := (#bYLS AND #iYLS.System_Error) OR (#bYLR AND ("LaserComm".Instance[#iInstance_Index].API.Inputs.YLR.Power_Supply_Alarm OR "LaserComm".Instance[#iInstance_Index].API.Inputs.YLR.Power_Supply_Failure));
END_REGION

REGION Network 27: Laser in Robot Mode Fault / Laser im Robotermodus-Fehler
   RUNG wire#powerrail
      Contact( #bYLS )
      I_Contact( #iYLS.Robot_Mode )
      wire#w1
      Coil( "LaserComm".Instance[#iInstance_Index].Scanner.Faults.%X21 )
   END_RUNG
   RUNG wire#powerrail
      Contact( #bYLR )
      I_Contact( "LaserComm".Instance[#iInstance_Index].API.Inputs.YLR.Keyswitch_in_REM_Position )
   END_RUNG wire#w1
   // the same network as SCL:
   "LaserComm".Instance[#iInstance_Index].Scanner.Faults.%X21 := (#bYLS AND NOT #iYLS.Robot_Mode) OR (#bYLR AND NOT "LaserComm".Instance[#iInstance_Index].API.Inputs.YLR.Keyswitch_in_REM_Position);
END_REGION

REGION Network 28: Laser Interlock Open Fault / Fehler Laserverriegelung offen
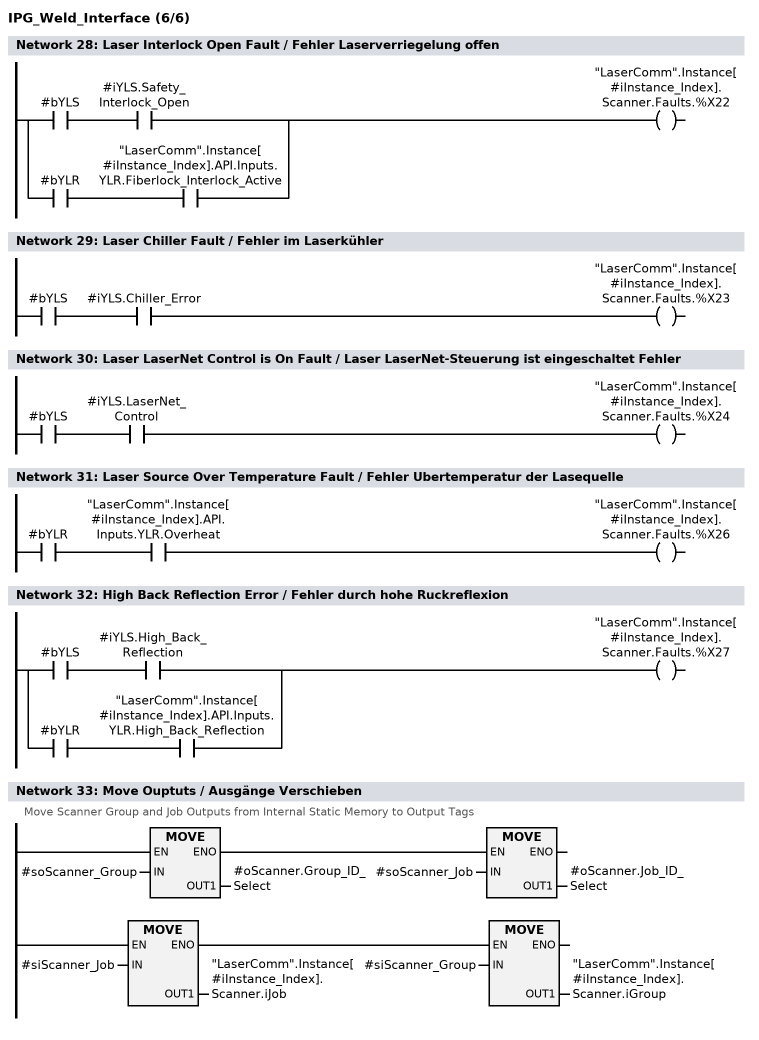
   RUNG wire#powerrail
      Contact( #bYLS )
      Contact( #iYLS.Safety_Interlock_Open )
      wire#w1
      Coil( "LaserComm".Instance[#iInstance_Index].Scanner.Faults.%X22 )
   END_RUNG
   RUNG wire#powerrail
      Contact( #bYLR )
      Contact( "LaserComm".Instance[#iInstance_Index].API.Inputs.YLR.Fiberlock_Interlock_Active )
   END_RUNG wire#w1
   // the same network as SCL:
   "LaserComm".Instance[#iInstance_Index].Scanner.Faults.%X22 := (#bYLS AND #iYLS.Safety_Interlock_Open) OR (#bYLR AND "LaserComm".Instance[#iInstance_Index].API.Inputs.YLR.Fiberlock_Interlock_Active);
END_REGION

REGION Network 29: Laser Chiller Fault / Fehler im Laserkühler
   RUNG wire#powerrail
      Contact( #bYLS )
      Contact( #iYLS.Chiller_Error )
      Coil( "LaserComm".Instance[#iInstance_Index].Scanner.Faults.%X23 )
   END_RUNG
   // the same network as SCL:
   "LaserComm".Instance[#iInstance_Index].Scanner.Faults.%X23 := #bYLS AND #iYLS.Chiller_Error;
END_REGION

REGION Network 30: Laser LaserNet Control is On Fault / Laser LaserNet-Steuerung ist eingeschaltet Fehler
   RUNG wire#powerrail
      Contact( #bYLS )
      Contact( #iYLS.LaserNet_Control )
      Coil( "LaserComm".Instance[#iInstance_Index].Scanner.Faults.%X24 )
   END_RUNG
   // the same network as SCL:
   "LaserComm".Instance[#iInstance_Index].Scanner.Faults.%X24 := #bYLS AND #iYLS.LaserNet_Control;
END_REGION

REGION Network 31: Laser Source Over Temperature Fault / Fehler Ubertemperatur der Lasequelle
   RUNG wire#powerrail
      Contact( #bYLR )
      Contact( "LaserComm".Instance[#iInstance_Index].API.Inputs.YLR.Overheat )
      Coil( "LaserComm".Instance[#iInstance_Index].Scanner.Faults.%X26 )
   END_RUNG
   // the same network as SCL:
   "LaserComm".Instance[#iInstance_Index].Scanner.Faults.%X26 := #bYLR AND "LaserComm".Instance[#iInstance_Index].API.Inputs.YLR.Overheat;
END_REGION

REGION Network 32: High Back Reflection Error / Fehler durch hohe Ruckreflexion
   RUNG wire#powerrail
      Contact( #bYLS )
      Contact( #iYLS.High_Back_Reflection )
      wire#w1
      Coil( "LaserComm".Instance[#iInstance_Index].Scanner.Faults.%X27 )
   END_RUNG
   RUNG wire#powerrail
      Contact( #bYLR )
      Contact( "LaserComm".Instance[#iInstance_Index].API.Inputs.YLR.High_Back_Reflection )
   END_RUNG wire#w1
   // the same network as SCL:
   "LaserComm".Instance[#iInstance_Index].Scanner.Faults.%X27 := (#bYLS AND #iYLS.High_Back_Reflection) OR (#bYLR AND "LaserComm".Instance[#iInstance_Index].API.Inputs.YLR.High_Back_Reflection);
END_REGION

REGION Network 33: Move Ouptuts / Ausgänge Verschieben
   // Move Scanner Group and Job Outputs from Internal Static Memory to Output Tags
   RUNG wire#powerrail
      Move(in := #soScanner_Group, out1 => #oScanner.Group_ID_Select)
      Move(in := #soScanner_Job, out1 => #oScanner.Job_ID_Select)
   END_RUNG
   RUNG wire#powerrail
      Move(in := #siScanner_Job, out1 => "LaserComm".Instance[#iInstance_Index].Scanner.iJob)
      Move(in := #siScanner_Group, out1 => "LaserComm".Instance[#iInstance_Index].Scanner.iGroup)
   END_RUNG
   // the same network as SCL:
   #oScanner.Group_ID_Select := #soScanner_Group;
   #oScanner.Job_ID_Select := #soScanner_Job;
   "LaserComm".Instance[#iInstance_Index].Scanner.iJob := #siScanner_Job;
   "LaserComm".Instance[#iInstance_Index].Scanner.iGroup := #siScanner_Group;
END_REGION
END_FUNCTION_BLOCK

FUNCTION_BLOCK "LaserComm_API"   // FB296, LAD
TITLE = LaserComm Communication Handling / SIS Communication Interface
{ S7_Optimized_Access := 'FALSE' }
VERSION : 2.0
// stored: AutoNumber true, IsIECCheckEnabled false, SetENOAutomatically false, UDAEnableTagReadback false
   VAR_INPUT
      iInstance_Index : Int;
      iSerial_Number : Array[1..32] of Char;
      iPart_Type : Array[1..18] of Char;
   END_VAR
   VAR DB_SPECIFIC
      sStep : Int;
      sLast_Step : Int;
      sReset : Bool;
      sLaserComm_Heart_Beat_F : Bool;
      sLaser_Heart_Beat_R : Bool;
      sHeartBeat_Dn : Bool;
      sHB_R { ExternalAccessible := 'False'; ExternalVisible := 'False'; ExternalWritable := 'False'} : Bool;
      sHB_F { ExternalAccessible := 'False'; ExternalVisible := 'False'; ExternalWritable := 'False'} : Bool;
      sLaserComm_Ready { ExternalAccessible := 'False'; ExternalVisible := 'False'; ExternalWritable := 'False'} : Bool;
      sReady_Reset : Bool;
      sLDD_Ref_Plane_Mismatch : Bool;
      sBlankResult : "LaserComm_LDD_Results";
      sBlankDDO { S7_SetPoint := 'True'} : "LaserComm_DDO";
      sData_MissMatch_Delay : IEC_TIMER;
      sStepTimeout : IEC_TIMER;
      sLaserComm_Heartbeat_Timer { S7_SetPoint := 'True'} : IEC_TIMER;
      sInstance_Inputs { S7_SetPoint := 'True'} : "API_Inputs";
      sInstance_Outputs { S7_SetPoint := 'True'} : "API_Outputs";
      sPointer : DInt;
      sHighest_Result : DInt;
   END_VAR
   VAR_TEMP
      tStep_Changed_ONS : Bool;
      tPointer : DInt;
   END_VAR
   // // sInstance_Inputs.Timeout : Timeout Value for API Job. Value set by Middleware and is dependant upon Job Function.
   VAR_TEMP   // added for the SCL form of the ladder/FBD networks
      _w1 : Bool;
      _w2 : Bool;
   END_VAR
BEGIN

REGION Network 1: Version
   // API Version
   // V1.1
   // Job Complete Flag Added to Step 30
   // Job Failed Fault Added
   // Over Pen Detection Disregarding Result Array if QA = 0
   // Move Instance Inputs and Outputs to Local Variables at Start and End of Block
   // V2
   // YLR Laser Type Supported
   // V3
   // Heart Beat Input Cleared Once Heart Beat Fault has Occurred
   // V4
   // Over Pen Bool Moved to LaserComm DB
   // Weld Mask added to LaserComm Outputs
   // Serial Number and Part Type added as inputs (Array of Chars)
   // General Tidy of Tags
   // Added Mutex
   // Added LDD Array Size constant and move to LaserComm DB register
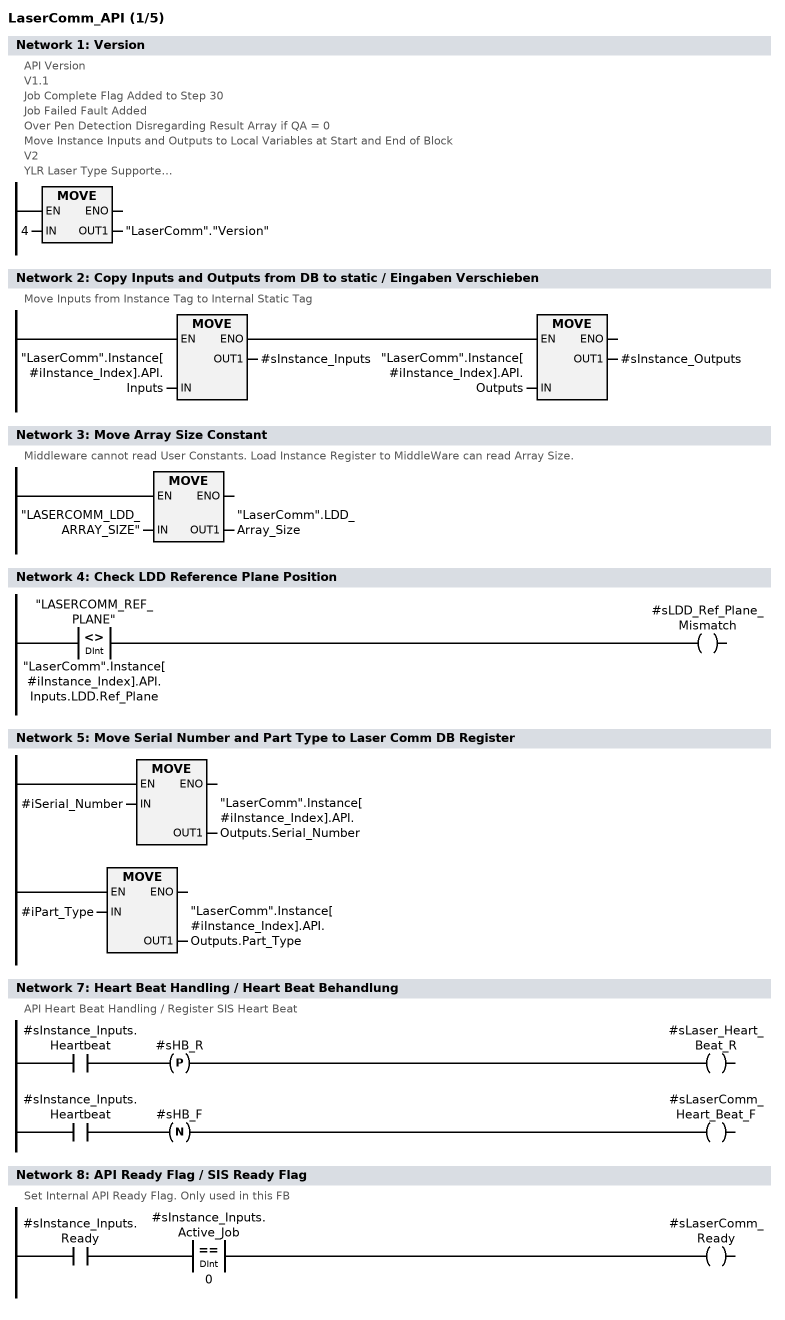
   RUNG wire#powerrail
      Move(in := 4, out1 => "LaserComm"."Version")
   END_RUNG
   // the same network as SCL:
   "LaserComm"."Version" := 4;
END_REGION

REGION Network 2: Copy Inputs and Outputs from DB to static / Eingaben Verschieben
   // Move Inputs from Instance Tag to Internal Static Tag
   RUNG wire#powerrail
      Move(in := "LaserComm".Instance[#iInstance_Index].API.Inputs, out1 => #sInstance_Inputs)
      Move(in := "LaserComm".Instance[#iInstance_Index].API.Outputs, out1 => #sInstance_Outputs)
   END_RUNG
   // the same network as SCL:
   #sInstance_Inputs := "LaserComm".Instance[#iInstance_Index].API.Inputs;
   #sInstance_Outputs := "LaserComm".Instance[#iInstance_Index].API.Outputs;
END_REGION

REGION Network 3: Move Array Size Constant
   // Middleware cannot read User Constants. Load Instance Register to MiddleWare can read Array Size.
   RUNG wire#powerrail
      Move(in := "LASERCOMM_LDD_ARRAY_SIZE", out1 => "LaserComm".LDD_Array_Size)
   END_RUNG
   // the same network as SCL:
   "LaserComm".LDD_Array_Size := "LASERCOMM_LDD_ARRAY_SIZE";
END_REGION

REGION Network 4: Check LDD Reference Plane Position
   RUNG wire#powerrail
      { S7_Templates := "SrcType := DInt" } NE_Contact(in1 := "LASERCOMM_REF_PLANE", in2 := "LaserComm".Instance[#iInstance_Index].API.Inputs.LDD.Ref_Plane)
      Coil( #sLDD_Ref_Plane_Mismatch )
   END_RUNG
   // the same network as SCL:
   #sLDD_Ref_Plane_Mismatch := "LASERCOMM_REF_PLANE" <> "LaserComm".Instance[#iInstance_Index].API.Inputs.LDD.Ref_Plane;
END_REGION

REGION Network 5: Move Serial Number and Part Type to Laser Comm DB Register
   RUNG wire#powerrail
      Move(in := #iSerial_Number, out1 => "LaserComm".Instance[#iInstance_Index].API.Outputs.Serial_Number)
   END_RUNG
   RUNG wire#powerrail
      Move(in := #iPart_Type, out1 => "LaserComm".Instance[#iInstance_Index].API.Outputs.Part_Type)
   END_RUNG
   // the same network as SCL:
   "LaserComm".Instance[#iInstance_Index].API.Outputs.Serial_Number := #iSerial_Number;
   "LaserComm".Instance[#iInstance_Index].API.Outputs.Part_Type := #iPart_Type;
END_REGION

REGION Network 6 (SCL): Over Penetration Detection / Erkennung Übermäßiger Penetration
   // Scan through the Results Array and Check for Over Penetration / Monitor QA_Results Array and look for Over Penetration Results Code
   // Monitor LDD QA Results and Check for Over Penetration
   //
   "LaserComm".Instance[#iInstance_Index].Static.OverPen_Detected := 0;

   FOR #tPointer := 0 TO "LASERCOMM_LDD_ARRAY_SIZE" DO
       IF #sInstance_Inputs.LDD.Results[#tPointer].QA <> 0 THEN
           IF #sInstance_Inputs.LDD.Results[#tPointer].Reasons.KHD.%X1 OR #sInstance_Inputs.LDD.Results[#tPointer].Reasons.KHD.%X2 THEN
               "LaserComm".Instance[#iInstance_Index].Static.OverPen_Detected := 1;
           END_IF;
       END_IF;
   END_FOR;
END_REGION

REGION Network 7: Heart Beat Handling / Heart Beat Behandlung
   // API Heart Beat Handling / Register SIS Heart Beat
   RUNG wire#powerrail
      Contact( #sInstance_Inputs.Heartbeat )
      P_Trig( #sHB_R )
      Coil( #sLaser_Heart_Beat_R )
   END_RUNG
   RUNG wire#powerrail
      Contact( #sInstance_Inputs.Heartbeat )
      N_Trig( #sHB_F )
      Coil( #sLaserComm_Heart_Beat_F )
   END_RUNG
   // the same network as SCL:
   #_w1 := #sInstance_Inputs.Heartbeat AND NOT #sHB_R;   // rising edge
   #sHB_R := #sInstance_Inputs.Heartbeat;
   #sLaser_Heart_Beat_R := #_w1;
   #_w2 := NOT #sInstance_Inputs.Heartbeat AND #sHB_F;   // falling edge
   #sHB_F := #sInstance_Inputs.Heartbeat;
   #sLaserComm_Heart_Beat_F := #_w2;
END_REGION

REGION Network 8: API Ready Flag / SIS Ready Flag
   // Set Internal API Ready Flag. Only used in this FB
   RUNG wire#powerrail
      Contact( #sInstance_Inputs.Ready )
      { S7_Templates := "SrcType := DInt" } EQ_Contact(in1 := #sInstance_Inputs.Active_Job, in2 := 0)
      Coil( #sLaserComm_Ready )
   END_RUNG
   // the same network as SCL:
   #sLaserComm_Ready := #sInstance_Inputs.Ready AND (#sInstance_Inputs.Active_Job = 0);
END_REGION

REGION Network 9: Step 0 / Schritt 0
   // Initial Step. Wait for IS Ready and Job Not Equal to 0. / Check SIS Ready, PLC Job is not 0 and PLC Start Job Is True
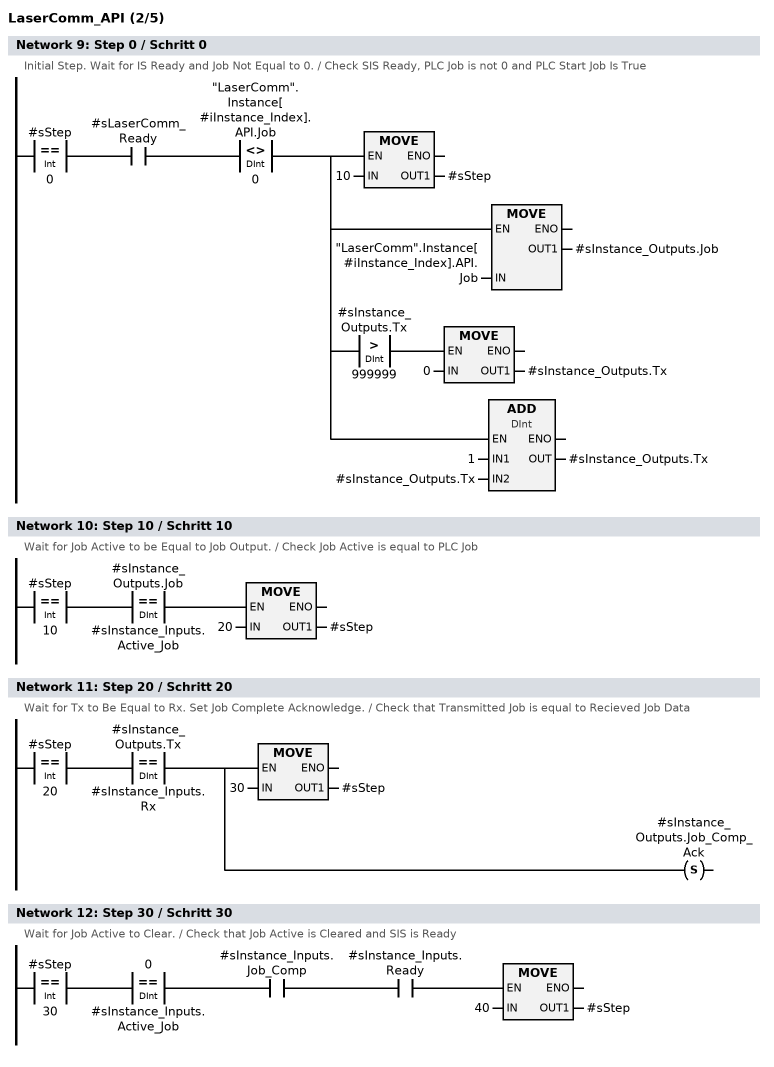
   RUNG wire#powerrail
      { S7_Templates := "SrcType := Int" } EQ_Contact(in1 := #sStep, in2 := 0)
      Contact( #sLaserComm_Ready )
      { S7_Templates := "SrcType := DInt" } NE_Contact(in1 := "LaserComm".Instance[#iInstance_Index].API.Job, in2 := 0)
      wire#w1
      { S7_GenerateENO := "TRUE" } Move(in := 10, out1 => #sStep)
   END_RUNG
   RUNG wire#w1
      { S7_GenerateENO := "TRUE" } Move(in := "LaserComm".Instance[#iInstance_Index].API.Job, out1 => #sInstance_Outputs.Job)
   END_RUNG
   RUNG wire#w1
      { S7_Templates := "SrcType := DInt" } GT_Contact(in1 := #sInstance_Outputs.Tx, in2 := 999999)
      { S7_GenerateENO := "TRUE" } Move(in := 0, out1 => #sInstance_Outputs.Tx)
   END_RUNG
   RUNG wire#w1
      { S7_Templates := "SrcType := DInt"; S7_GenerateENO := "TRUE" } Add(in1 := 1, in2 := #sInstance_Outputs.Tx, out => #sInstance_Outputs.Tx)
   END_RUNG
   // the same network as SCL:
   #_w1 := (#sStep = 0) AND #sLaserComm_Ready AND ("LaserComm".Instance[#iInstance_Index].API.Job <> 0);
   IF #_w1 THEN
       #sStep := 10;
       #sInstance_Outputs.Job := "LaserComm".Instance[#iInstance_Index].API.Job;
   END_IF;
   IF #_w1 AND (#sInstance_Outputs.Tx > 999999) THEN #sInstance_Outputs.Tx := 0; END_IF;
   IF #_w1 THEN #sInstance_Outputs.Tx := 1 + #sInstance_Outputs.Tx; END_IF;
END_REGION

REGION Network 10: Step 10 / Schritt 10
   // Wait for Job Active to be Equal to Job Output. / Check Job Active is equal to PLC Job
   RUNG wire#powerrail
      { S7_Templates := "SrcType := Int" } EQ_Contact(in1 := #sStep, in2 := 10)
      { S7_Templates := "SrcType := DInt" } EQ_Contact(in1 := #sInstance_Outputs.Job, in2 := #sInstance_Inputs.Active_Job)
      { S7_GenerateENO := "TRUE" } Move(in := 20, out1 => #sStep)
   END_RUNG
   // the same network as SCL:
   IF (#sStep = 10) AND (#sInstance_Outputs.Job = #sInstance_Inputs.Active_Job) THEN #sStep := 20; END_IF;
END_REGION

REGION Network 11: Step 20 / Schritt 20
   // Wait for Tx to Be Equal to Rx. Set Job Complete Acknowledge. / Check that Transmitted Job is equal to Recieved Job Data
   RUNG wire#powerrail
      { S7_Templates := "SrcType := Int" } EQ_Contact(in1 := #sStep, in2 := 20)
      { S7_Templates := "SrcType := DInt" } EQ_Contact(in1 := #sInstance_Outputs.Tx, in2 := #sInstance_Inputs.Rx)
      wire#w1
      { S7_GenerateENO := "TRUE" } Move(in := 30, out1 => #sStep)
   END_RUNG
   RUNG wire#w1
      S_Coil( #sInstance_Outputs.Job_Comp_Ack )
   END_RUNG
   // the same network as SCL:
   #_w1 := (#sStep = 20) AND (#sInstance_Outputs.Tx = #sInstance_Inputs.Rx);
   IF #_w1 THEN
       #sStep := 30;
       #sInstance_Outputs.Job_Comp_Ack := TRUE;
   END_IF;
END_REGION

REGION Network 12: Step 30 / Schritt 30
   // Wait for Job Active to Clear. / Check that Job Active is Cleared and SIS is Ready
   RUNG wire#powerrail
      { S7_Templates := "SrcType := Int" } EQ_Contact(in1 := #sStep, in2 := 30)
      { S7_Templates := "SrcType := DInt" } EQ_Contact(in1 := 0, in2 := #sInstance_Inputs.Active_Job)
      Contact( #sInstance_Inputs.Job_Comp )
      Contact( #sInstance_Inputs.Ready )
      { S7_GenerateENO := "TRUE" } Move(in := 40, out1 => #sStep)
   END_RUNG
   // the same network as SCL:
   IF (#sStep = 30) AND (0 = #sInstance_Inputs.Active_Job) AND #sInstance_Inputs.Job_Comp AND #sInstance_Inputs.Ready THEN
       #sStep := 40;
   END_IF;
END_REGION

REGION Network 13: Step 40 / Schritt 40
   // Reset Step
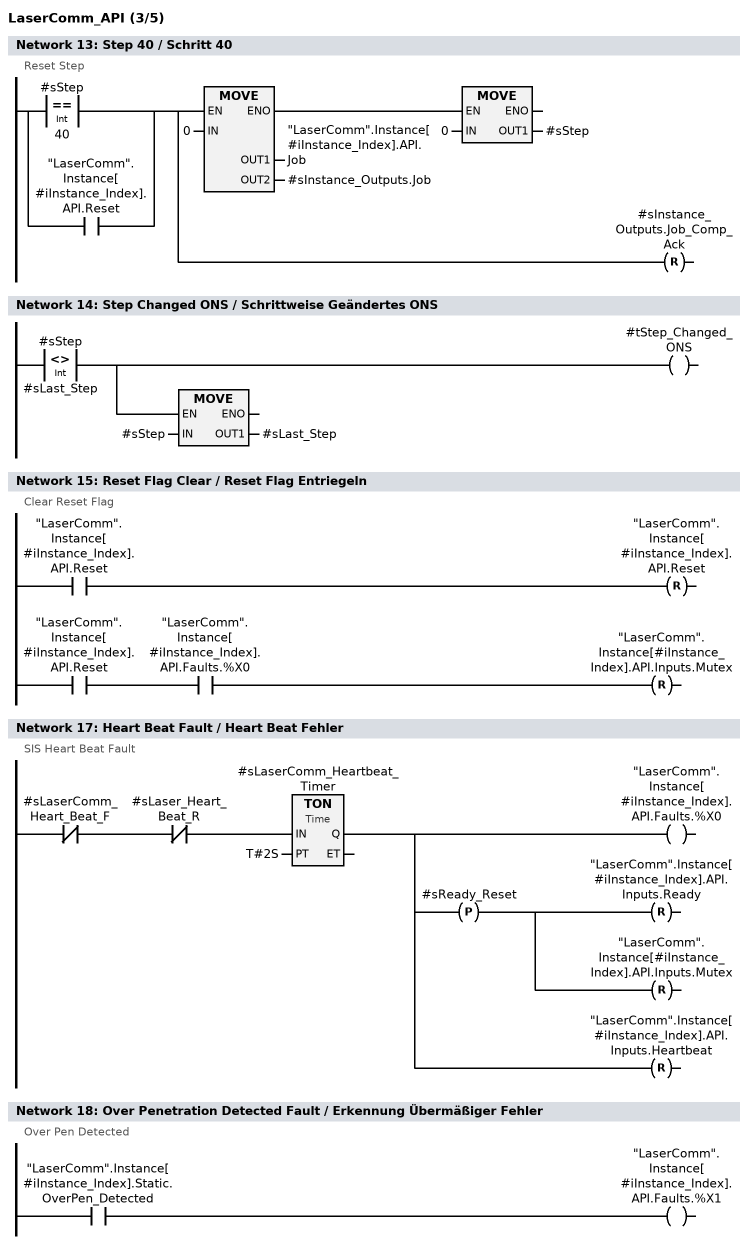
   RUNG wire#powerrail
      { S7_Templates := "SrcType := Int" } EQ_Contact(in1 := #sStep, in2 := 40)
      wire#w1
      { S7_GenerateENO := "TRUE" } Move(in := 0, out1 => "LaserComm".Instance[#iInstance_Index].API.Job, out2 => #sInstance_Outputs.Job)
      { S7_GenerateENO := "TRUE" } Move(in := 0, out1 => #sStep)
   END_RUNG
   RUNG wire#powerrail
      Contact( "LaserComm".Instance[#iInstance_Index].API.Reset )
   END_RUNG wire#w1
   RUNG wire#w1
      R_Coil( #sInstance_Outputs.Job_Comp_Ack )
   END_RUNG
   // the same network as SCL:
   // ENO of a box is taken as its EN; it also drops when the box reports an error
   #_w1 := (#sStep = 40) OR "LaserComm".Instance[#iInstance_Index].API.Reset;
   #_w2 := (#sStep = 40) OR "LaserComm".Instance[#iInstance_Index].API.Reset;
   IF #_w2 THEN
       "LaserComm".Instance[#iInstance_Index].API.Job := 0;
       #sInstance_Outputs.Job := 0;
       #sStep := 0;
   END_IF;
   IF #_w1 THEN #sInstance_Outputs.Job_Comp_Ack := FALSE; END_IF;
END_REGION

REGION Network 14: Step Changed ONS / Schrittweise Geändertes ONS
   RUNG wire#powerrail
      { S7_Templates := "SrcType := Int" } NE_Contact(in1 := #sStep, in2 := #sLast_Step)
      wire#w1
      Coil( #tStep_Changed_ONS )
   END_RUNG
   RUNG wire#w1
      { S7_GenerateENO := "TRUE" } Move(in := #sStep, out1 => #sLast_Step)
   END_RUNG
   // the same network as SCL:
   #tStep_Changed_ONS := #sStep <> #sLast_Step;
   IF #tStep_Changed_ONS THEN #sLast_Step := #sStep; END_IF;
END_REGION

REGION Network 15: Reset Flag Clear / Reset Flag Entriegeln
   // Clear Reset Flag
   RUNG wire#powerrail
      Contact( "LaserComm".Instance[#iInstance_Index].API.Reset )
      R_Coil( "LaserComm".Instance[#iInstance_Index].API.Reset )
   END_RUNG
   RUNG wire#powerrail
      Contact( "LaserComm".Instance[#iInstance_Index].API.Reset )
      Contact( "LaserComm".Instance[#iInstance_Index].API.Faults.%X0 )
      R_Coil( "LaserComm".Instance[#iInstance_Index].API.Inputs.Mutex )
   END_RUNG
   // the same network as SCL:
   IF "LaserComm".Instance[#iInstance_Index].API.Reset THEN
       "LaserComm".Instance[#iInstance_Index].API.Reset := FALSE;
   END_IF;
   IF "LaserComm".Instance[#iInstance_Index].API.Reset AND "LaserComm".Instance[#iInstance_Index].API.Faults.%X0 THEN
       "LaserComm".Instance[#iInstance_Index].API.Inputs.Mutex := FALSE;
   END_IF;
END_REGION

REGION Network 16 (SCL): Clear Results Array / Ergebnis-Array Löschen
   // Clear the Results Array

   IF #sInstance_Inputs.Clear_Results THEN
       FOR #tPointer := 0 TO "LASERCOMM_LDD_ARRAY_SIZE" DO
           "LaserComm".Instance[#iInstance_Index].API.Inputs.LDD.Results[#tPointer] := #sBlankResult;
           "LaserComm".Instance[#iInstance_Index].API.Inputs.LDD.DDO[#tPointer] := #sBlankDDO;
       END_FOR;
   END_IF;

   "LaserComm".Instance[#iInstance_Index].API.Inputs.Clear_Results := FALSE;
END_REGION

REGION Network 17: Heart Beat Fault / Heart Beat Fehler
   // SIS Heart Beat Fault
   RUNG wire#powerrail
      I_Contact( #sLaserComm_Heart_Beat_F )
      I_Contact( #sLaser_Heart_Beat_R )
      { S7_Templates := "time_type := Time" } #sLaserComm_Heartbeat_Timer.TON(pt := T#2S, et =>)
      wire#w1
      Coil( "LaserComm".Instance[#iInstance_Index].API.Faults.%X0 )
   END_RUNG
   RUNG wire#w1
      P_Trig( #sReady_Reset )
      wire#w2
      R_Coil( "LaserComm".Instance[#iInstance_Index].API.Inputs.Ready )
   END_RUNG
   RUNG wire#w2
      R_Coil( "LaserComm".Instance[#iInstance_Index].API.Inputs.Mutex )
   END_RUNG
   RUNG wire#w1
      R_Coil( "LaserComm".Instance[#iInstance_Index].API.Inputs.Heartbeat )
   END_RUNG
   // the same network as SCL:
   #sLaserComm_Heartbeat_Timer.TON(IN := NOT #sLaserComm_Heart_Beat_F AND NOT #sLaser_Heart_Beat_R, PT := T#2S);
   "LaserComm".Instance[#iInstance_Index].API.Faults.%X0 := #sLaserComm_Heartbeat_Timer.Q;
   #_w1 := #sLaserComm_Heartbeat_Timer.Q AND NOT #sReady_Reset;   // rising edge
   #sReady_Reset := #sLaserComm_Heartbeat_Timer.Q;
   IF #_w1 THEN
       "LaserComm".Instance[#iInstance_Index].API.Inputs.Ready := FALSE;
       "LaserComm".Instance[#iInstance_Index].API.Inputs.Mutex := FALSE;
   END_IF;
   IF #sLaserComm_Heartbeat_Timer.Q THEN
       "LaserComm".Instance[#iInstance_Index].API.Inputs.Heartbeat := FALSE;
   END_IF;
END_REGION

REGION Network 18: Over Penetration Detected Fault / Erkennung Übermäßiger Fehler
   // Over Pen Detected
   RUNG wire#powerrail
      Contact( "LaserComm".Instance[#iInstance_Index].Static.OverPen_Detected )
      Coil( "LaserComm".Instance[#iInstance_Index].API.Faults.%X1 )
   END_RUNG
   // the same network as SCL:
   "LaserComm".Instance[#iInstance_Index].API.Faults.%X1 := "LaserComm".Instance[#iInstance_Index].Static.OverPen_Detected;
END_REGION

REGION Network 19: Sequence Timeout Fault / Sequenz Timeout Fehler
   // SIS Command has taken too long to complete. PT Value set by SIS.
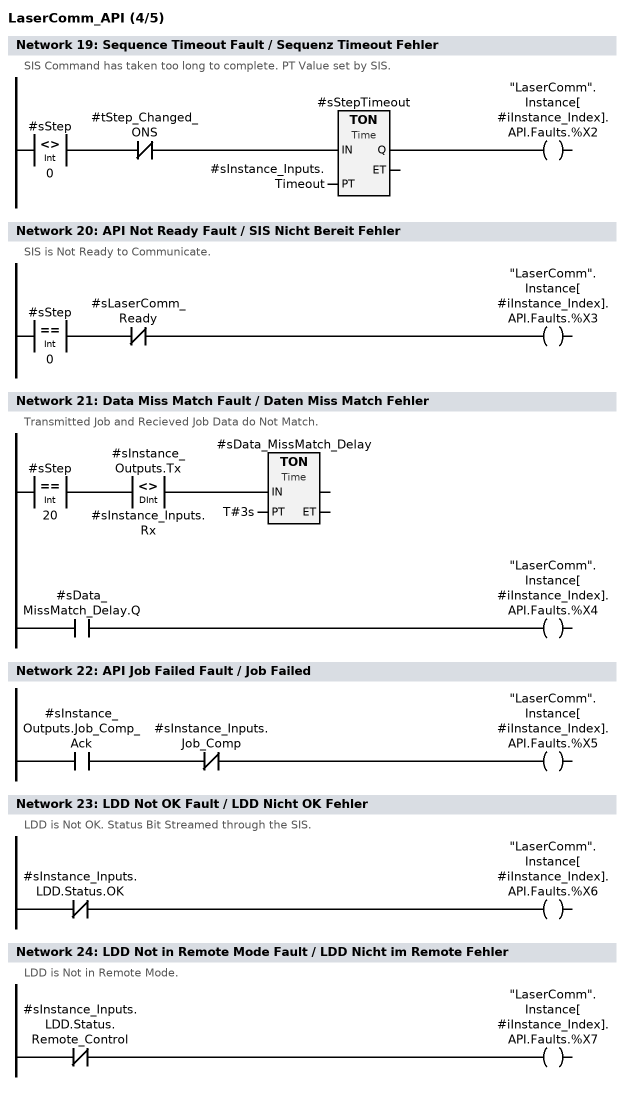
   RUNG wire#powerrail
      { S7_Templates := "SrcType := Int" } NE_Contact(in1 := #sStep, in2 := 0)
      I_Contact( #tStep_Changed_ONS )
      { S7_Templates := "time_type := Time" } #sStepTimeout.TON(pt := #sInstance_Inputs.Timeout, et =>)
      Coil( "LaserComm".Instance[#iInstance_Index].API.Faults.%X2 )
   END_RUNG
   // the same network as SCL:
   #sStepTimeout.TON(IN := (#sStep <> 0) AND NOT #tStep_Changed_ONS, PT := #sInstance_Inputs.Timeout);
   "LaserComm".Instance[#iInstance_Index].API.Faults.%X2 := #sStepTimeout.Q;
END_REGION

REGION Network 20: API Not Ready Fault / SIS Nicht Bereit Fehler
   // SIS is Not Ready to Communicate.
   RUNG wire#powerrail
      { S7_Templates := "SrcType := Int" } EQ_Contact(in1 := #sStep, in2 := 0)
      I_Contact( #sLaserComm_Ready )
      Coil( "LaserComm".Instance[#iInstance_Index].API.Faults.%X3 )
   END_RUNG
   // the same network as SCL:
   "LaserComm".Instance[#iInstance_Index].API.Faults.%X3 := (#sStep = 0) AND NOT #sLaserComm_Ready;
END_REGION

REGION Network 21: Data Miss Match Fault / Daten Miss Match Fehler
   // Transmitted Job and Recieved Job Data do Not Match.
   RUNG wire#powerrail
      { S7_Templates := "SrcType := Int" } EQ_Contact(in1 := #sStep, in2 := 20)
      { S7_Templates := "SrcType := DInt" } NE_Contact(in1 := #sInstance_Outputs.Tx, in2 := #sInstance_Inputs.Rx)
      { S7_Templates := "time_type := Time" } #sData_MissMatch_Delay.TON(pt := T#3s, et =>)
   END_RUNG
   RUNG wire#powerrail
      Contact( #sData_MissMatch_Delay.Q )
      Coil( "LaserComm".Instance[#iInstance_Index].API.Faults.%X4 )
   END_RUNG
   // the same network as SCL:
   #sData_MissMatch_Delay.TON(IN := (#sStep = 20) AND (#sInstance_Outputs.Tx <> #sInstance_Inputs.Rx),
                           PT := T#3s);
   "LaserComm".Instance[#iInstance_Index].API.Faults.%X4 := #sData_MissMatch_Delay.Q;
END_REGION

REGION Network 22: API Job Failed Fault / Job Failed
   RUNG wire#powerrail
      Contact( #sInstance_Outputs.Job_Comp_Ack )
      I_Contact( #sInstance_Inputs.Job_Comp )
      Coil( "LaserComm".Instance[#iInstance_Index].API.Faults.%X5 )
   END_RUNG
   // the same network as SCL:
   "LaserComm".Instance[#iInstance_Index].API.Faults.%X5 := #sInstance_Outputs.Job_Comp_Ack AND NOT #sInstance_Inputs.Job_Comp;
END_REGION

REGION Network 23: LDD Not OK Fault / LDD Nicht OK Fehler
   // LDD is Not OK. Status Bit Streamed through the SIS.
   RUNG wire#powerrail
      I_Contact( #sInstance_Inputs.LDD.Status.OK )
      Coil( "LaserComm".Instance[#iInstance_Index].API.Faults.%X6 )
   END_RUNG
   // the same network as SCL:
   "LaserComm".Instance[#iInstance_Index].API.Faults.%X6 := NOT #sInstance_Inputs.LDD.Status.OK;
END_REGION

REGION Network 24: LDD Not in Remote Mode Fault / LDD Nicht im Remote Fehler
   // LDD is Not in Remote Mode.
   RUNG wire#powerrail
      I_Contact( #sInstance_Inputs.LDD.Status.Remote_Control )
      Coil( "LaserComm".Instance[#iInstance_Index].API.Faults.%X7 )
   END_RUNG
   // the same network as SCL:
   "LaserComm".Instance[#iInstance_Index].API.Faults.%X7 := NOT #sInstance_Inputs.LDD.Status.Remote_Control;
END_REGION

REGION Network 25: LDD Reference Plane Mismatch Fault / LDD Nicht im Remote Fehler
   // LDD is Not in Remote Mode.
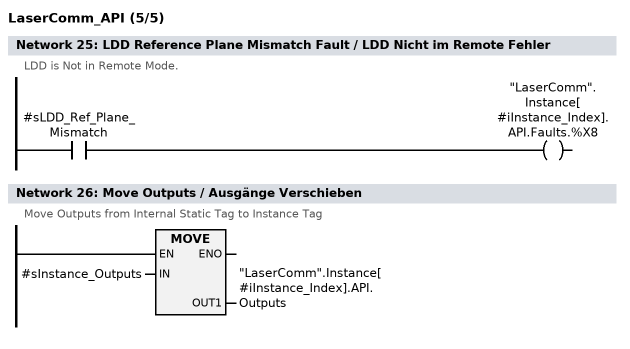
   RUNG wire#powerrail
      Contact( #sLDD_Ref_Plane_Mismatch )
      Coil( "LaserComm".Instance[#iInstance_Index].API.Faults.%X8 )
   END_RUNG
   // the same network as SCL:
   "LaserComm".Instance[#iInstance_Index].API.Faults.%X8 := #sLDD_Ref_Plane_Mismatch;
END_REGION

REGION Network 26: Move Outputs / Ausgänge Verschieben
   // Move Outputs from Internal Static Tag to Instance Tag
   RUNG wire#powerrail
      Move(in := #sInstance_Outputs, out1 => "LaserComm".Instance[#iInstance_Index].API.Outputs)
   END_RUNG
   // the same network as SCL:
   "LaserComm".Instance[#iInstance_Index].API.Outputs := #sInstance_Outputs;
END_REGION
END_FUNCTION_BLOCK

DATA_BLOCK "Call_DB"   // DB7
VERSION : 0.1
// stored: AutoNumber true, DBAccessibleFromOPCUA true, DBAccessibleFromWebserver true, InstanceOfName Call, InstanceOfType FB
"Call"
BEGIN
END_DATA_BLOCK

DATA_BLOCK "Control_DB"   // DB2
VERSION : 0.1
// stored: AutoNumber true, DBAccessibleFromOPCUA true, DBAccessibleFromWebserver true, InstanceOfName Control, InstanceOfType FB
"Control"
BEGIN
END_DATA_BLOCK

DATA_BLOCK "Graph_Sequence_DB"   // DB3
VERSION : 0.1
// stored: AutoNumber true, DBAccessibleFromOPCUA true, DBAccessibleFromWebserver true, InstanceOfName Graph_Sequence, InstanceOfType FB
"Graph_Sequence"
BEGIN
END_DATA_BLOCK

DATA_BLOCK "IPG_Weld_Interface_DB"   // DB4
VERSION : 1.0
// stored: AutoNumber true, DBAccessibleFromOPCUA true, DBAccessibleFromWebserver true, InstanceOfName IPG_Weld_Interface, InstanceOfType FB
"IPG_Weld_Interface"
BEGIN
END_DATA_BLOCK
